KUKA KRL program: MyProgram_007().src

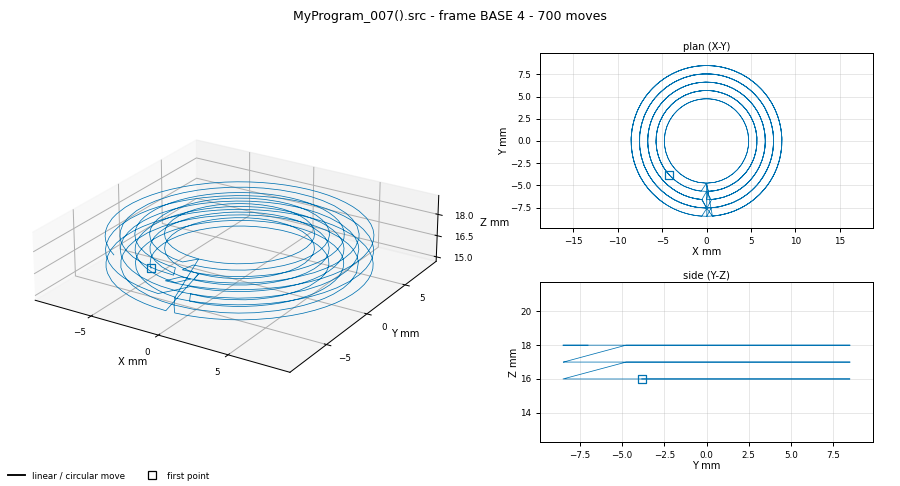
[picture p0: tool path of MyProgram_007().src in frame BASE 4, 700 of 700 moves have a stored position in this frame; points joined in program order, loops and branches not executed]
&ACCESS RVP
&REL 1
&PARAM TEMPLATE = C:\KRC\Roboter\Template\vorgabe
&PARAM EDITMASK = *
DEF MyProgram_007()
; ---- Setting reference (Base) ----
$BASE = BASE_DATA[4]

; --------------------------
; ---- Setting tool (TCP) ----
$TOOL = TOOL_DATA[3]
; --------------------------

$VEL.CP = VEL_APROX_PRINT
Startdeposition()
$VEL.CP = VEL_PRINT
LIN {X -4.1993,Y -3.8325,Z 16,A -3.0897,B 0,C 0,E1 0.1598,E2 90.0712} C_DIS
LIN {X -4.6903,Y -3.2125,Z 16,A -3.0815,B 0,C 0,E1 0.1598,E2 90.0712} C_DIS
LIN {X -5.0898,Y -2.5301,Z 16,A -3.0673,B 0,C 0,E1 0.1598,E2 90.0712} C_DIS
LIN {X -5.3905,Y -1.7989,Z 16,A -3.0475,B 0,C 0,E1 0.1598,E2 90.0712} C_DIS
LIN {X -5.5883,Y -1.0336,Z 16,A -3.0224,B 0,C 0,E1 0.1598,E2 90.0712} C_DIS
LIN {X -5.6777,Y -0.2482,Z 16,A -2.9925,B 0,C 0,E1 0.1598,E2 90.0712} C_DIS
LIN {X -5.6569,Y 0.542,Z 16,A -2.9584,B 0,C 0,E1 0.1598,E2 90.0713} C_DIS
LIN {X -5.5287,Y 1.3221,Z 16,A -2.9208,B 0,C 0,E1 0.1598,E2 90.0713} C_DIS
LIN {X -5.293,Y 2.077,Z 16,A -2.8803,B 0,C 0,E1 0.1598,E2 90.0714} C_DIS
LIN {X -4.954,Y 2.7915,Z 16,A -2.8378,B 0,C 0,E1 0.1598,E2 90.0715} C_DIS
LIN {X -4.5175,Y 3.4508,Z 16,A -2.7939,B 0,C 0,E1 0.1598,E2 90.0716} C_DIS
LIN {X -3.9945,Y 4.044,Z 16,A -2.7497,B 0,C 0,E1 0.1598,E2 90.0717} C_DIS
LIN {X -3.395,Y 4.5593,Z 16,A -2.7059,B 0,C 0,E1 0.1598,E2 90.0718} C_DIS
LIN {X -2.7289,Y 4.9855,Z 16,A -2.6634,B 0,C 0,E1 0.1598,E2 90.0719} C_DIS
LIN {X -2.0108,Y 5.316,Z 16,A -2.623,B 0,C 0,E1 0.1598,E2 90.072} C_DIS
LIN {X -1.2535,Y 5.5427,Z 16,A -2.5855,B 0,C 0,E1 0.1598,E2 90.0721} C_DIS
LIN {X -0.2754,Y 5.684,Z 16,A -2.5435,B 0,C 0,E1 0.1598,E2 90.0721} C_DIS
LIN {X 0.4673,Y 5.6661,Z 16,A -2.5168,B 0,C 0,E1 0.1598,E2 90.0722} C_DIS
LIN {X 1.1226,Y 5.5779,Z 16,A -2.4964,B 0,C 0,E1 0.1598,E2 90.0722} C_DIS
LIN {X 2.1788,Y 5.2504,Z 16,A -2.4712,B 0,C 0,E1 0.1598,E2 90.0722} C_DIS
LIN {X 2.8813,Y 4.8983,Z 16,A -2.4602,B 0,C 0,E1 0.1598,E2 90.0722} C_DIS
LIN {X 3.5298,Y 4.4549,Z 16,A -2.455,B 0,C 0,E1 0.1598,E2 90.0722} C_DIS
LIN {X 4.1099,Y 3.9251,Z 16,A -2.456,B 0,C 0,E1 0.1598,E2 90.0722} C_DIS
LIN {X 4.6118,Y 3.3208,Z 16,A -2.4631,B 0,C 0,E1 0.1598,E2 90.0721} C_DIS
LIN {X 5.0254,Y 2.653,Z 16,A -2.4761,B 0,C 0,E1 0.1598,E2 90.0721} C_DIS
LIN {X 5.3429,Y 1.9345,Z 16,A -2.4949,B 0,C 0,E1 0.1598,E2 90.0719} C_DIS
LIN {X 5.5612,Y 1.1798,Z 16,A -2.5188,B 0,C 0,E1 0.1598,E2 90.0719} C_DIS
LIN {X 5.6718,Y 0.4017,Z 16,A -2.5478,B 0,C 0,E1 0.1598,E2 90.0719} C_DIS
LIN {X 5.6312,Y -0.8177,Z 16,A -2.6006,B 0,C 0,E1 0.1598,E2 90.0713} C_DIS
LIN {X 5.4243,Y -1.7083,Z 16,A -2.6464,B 0,C 0,E1 0.1598,E2 90.0716} C_DIS
LIN {X 5.159,Y -2.3898,Z 16,A -2.6852,B 0,C 0,E1 0.1598,E2 90.0717} C_DIS
LIN {X 4.8093,Y -3.0322,Z 16,A -2.7254,B 0,C 0,E1 0.1598,E2 90.0717} C_DIS
LIN {X 4.3781,Y -3.6227,Z 16,A -2.7663,B 0,C 0,E1 0.1598,E2 90.0717} C_DIS
LIN {X 3.8775,Y -4.1555,Z 16,A -2.8073,B 0,C 0,E1 0.1598,E2 90.0717} C_DIS
LIN {X 3.3125,Y -4.6195,Z 16,A -2.8478,B 0,C 0,E1 0.1598,E2 90.0717} C_DIS
LIN {X 2.287,Y -5.2099,Z 16,A -2.9105,B 0,C 0,E1 0.1598,E2 90.0715} C_DIS
LIN {X 1.4913,Y -5.4882,Z 16,A -2.9516,B 0,C 0,E1 0.1598,E2 90.0716} C_DIS
LIN {X 0.8312,Y -5.6248,Z 16,A -2.9816,B 0,C 0,E1 0.1598,E2 90.0716} C_DIS
LIN {X -0.0092,Y -5.6859,Z 16,A -3.0151,B 0,C 0,E1 0.1598,E2 90.0716} C_DIS
Enddeposition()
LIN {X -0.0092,Y -5.6859,Z 16,A -3.0151,B 0,C 0,E1 0.1598,E2 90.0716} C_DIS
Startdeposition()
$VEL.CP = VEL_PRINT
LIN {X 0.5176,Y -6.5991,Z 16,A -3.034,B 0,C 0,E1 0.1598,E2 90.071} C_DIS
LIN {X 1.2141,Y -6.5071,Z 16,A -3.0051,B 0,C 0,E1 0.1598,E2 90.0715} C_DIS
LIN {X 1.897,Y -6.3414,Z 16,A -2.9731,B 0,C 0,E1 0.1598,E2 90.0715} C_DIS
LIN {X 2.5586,Y -6.1047,Z 16,A -2.9387,B 0,C 0,E1 0.1598,E2 90.0716} C_DIS
LIN {X 3.1928,Y -5.802,Z 16,A -2.9026,B 0,C 0,E1 0.1598,E2 90.0716} C_DIS
LIN {X 3.7886,Y -5.4294,Z 16,A -2.8649,B 0,C 0,E1 0.1598,E2 90.0716} C_DIS
LIN {X 4.3414,Y -4.9954,Z 16,A -2.8261,B 0,C 0,E1 0.1598,E2 90.0717} C_DIS
LIN {X 4.8479,Y -4.5083,Z 16,A -2.7868,B 0,C 0,E1 0.1598,E2 90.0717} C_DIS
LIN {X 5.2989,Y -3.9693,Z 16,A -2.7473,B 0,C 0,E1 0.1598,E2 90.0717} C_DIS
LIN {X 5.6898,Y -3.3855,Z 16,A -2.7081,B 0,C 0,E1 0.1598,E2 90.0717} C_DIS
LIN {X 6.0154,Y -2.7628,Z 16,A -2.6697,B 0,C 0,E1 0.1598,E2 90.0718} C_DIS
LIN {X 6.2743,Y -2.1096,Z 16,A -2.6324,B 0,C 0,E1 0.1598,E2 90.0718} C_DIS
LIN {X 6.4633,Y -1.4327,Z 16,A -2.5967,B 0,C 0,E1 0.1598,E2 90.0718} C_DIS
LIN {X 6.5765,Y -0.7393,Z 16,A -2.563,B 0,C 0,E1 0.1598,E2 90.0718} C_DIS
LIN {X 6.6202,Y -0.038,Z 16,A -2.5316,B 0,C 0,E1 0.1598,E2 90.0719} C_DIS
LIN {X 6.5859,Y 0.6639,Z 16,A -2.5031,B 0,C 0,E1 0.1598,E2 90.0719} C_DIS
LIN {X 6.4813,Y 1.3587,Z 16,A -2.4774,B 0,C 0,E1 0.1598,E2 90.0719} C_DIS
LIN {X 6.2989,Y 2.0375,Z 16,A -2.4553,B 0,C 0,E1 0.1598,E2 90.072} C_DIS
LIN {X 6.0478,Y 2.6938,Z 16,A -2.4367,B 0,C 0,E1 0.1598,E2 90.072} C_DIS
LIN {X 5.7274,Y 3.3193,Z 16,A -2.422,B 0,C 0,E1 0.1598,E2 90.0721} C_DIS
LIN {X 5.3436,Y 3.908,Z 16,A -2.4112,B 0,C 0,E1 0.1598,E2 90.0721} C_DIS
LIN {X 4.8987,Y 4.4518,Z 16,A -2.4046,B 0,C 0,E1 0.1598,E2 90.0721} C_DIS
LIN {X 4.3987,Y 4.9454,Z 16,A -2.4021,B 0,C 0,E1 0.1598,E2 90.0722} C_DIS
LIN {X 3.8499,Y 5.3843,Z 16,A -2.4038,B 0,C 0,E1 0.1598,E2 90.0722} C_DIS
LIN {X 2.9549,Y 5.9276,Z 16,A -2.4138,B 0,C 0,E1 0.1598,E2 90.0722} C_DIS
LIN {X 2.1433,Y 6.2629,Z 16,A -2.4296,B 0,C 0,E1 0.1598,E2 90.0722} C_DIS
LIN {X 1.4674,Y 6.4547,Z 16,A -2.4465,B 0,C 0,E1 0.1598,E2 90.0722} C_DIS
LIN {X 0.7748,Y 6.5728,Z 16,A -2.4671,B 0,C 0,E1 0.1598,E2 90.0722} C_DIS
LIN {X 0.0739,Y 6.6206,Z 16,A -2.4909,B 0,C 0,E1 0.1598,E2 90.0722} C_DIS
LIN {X -0.6281,Y 6.5907,Z 16,A -2.5181,B 0,C 0,E1 0.1598,E2 90.0722} C_DIS
LIN {X -1.3232,Y 6.4884,Z 16,A -2.5481,B 0,C 0,E1 0.1598,E2 90.0722} C_DIS
LIN {X -2.0031,Y 6.3109,Z 16,A -2.5806,B 0,C 0,E1 0.1598,E2 90.0722} C_DIS
LIN {X -2.6597,Y 6.0605,Z 16,A -2.6154,B 0,C 0,E1 0.1598,E2 90.0721} C_DIS
LIN {X -3.2875,Y 5.7451,Z 16,A -2.6518,B 0,C 0,E1 0.1598,E2 90.072} C_DIS
LIN {X -3.8778,Y 5.3647,Z 16,A -2.6896,B 0,C 0,E1 0.1598,E2 90.072} C_DIS
LIN {X -4.4251,Y 4.924,Z 16,A -2.7284,B 0,C 0,E1 0.1598,E2 90.0718} C_DIS
LIN {X -4.921,Y 4.4263,Z 16,A -2.7676,B 0,C 0,E1 0.1598,E2 90.0718} C_DIS
LIN {X -5.3638,Y 3.8808,Z 16,A -2.8069,B 0,C 0,E1 0.1598,E2 90.0717} C_DIS
LIN {X -5.745,Y 3.2907,Z 16,A -2.8458,B 0,C 0,E1 0.1598,E2 90.0717} C_DIS
LIN {X -6.0618,Y 2.6636,Z 16,A -2.8839,B 0,C 0,E1 0.1598,E2 90.0715} C_DIS
LIN {X -6.3071,Y 2.0053,Z 16,A -2.9206,B 0,C 0,E1 0.1598,E2 90.0715} C_DIS
LIN {X -6.4853,Y 1.3257,Z 16,A -2.9558,B 0,C 0,E1 0.1598,E2 90.0714} C_DIS
LIN {X -6.59,Y 0.631,Z 16,A -2.9889,B 0,C 0,E1 0.1598,E2 90.0714} C_DIS
LIN {X -6.6205,Y -0.0711,Z 16,A -3.0196,B 0,C 0,E1 0.1598,E2 90.0713} C_DIS
LIN {X -6.5747,Y -0.7722,Z 16,A -3.0475,B 0,C 0,E1 0.1598,E2 90.0713} C_DIS
LIN {X -6.4566,Y -1.4648,Z 16,A -3.0724,B 0,C 0,E1 0.1598,E2 90.0713} C_DIS
LIN {X -6.2639,Y -2.1405,Z 16,A -3.0938,B 0,C 0,E1 0.1598,E2 90.0713} C_DIS
LIN {X -6.001,Y -2.7921,Z 16,A -3.1116,B 0,C 0,E1 0.1598,E2 90.0713} C_DIS
LIN {X -5.5827,Y -3.5644,Z 16,A -3.1287,B 0,C 0,E1 0.1598,E2 90.071} C_DIS
LIN {X -4.9457,Y -4.3995,Z 16,A -3.1406,B 0,C 0,E1 0.1598,E2 90.071} C_DIS
LIN {X -4.4386,Y -4.9094,Z 16,A -3.1437,B 0,C 0,E1 0.1598,E2 90.0712} C_DIS
LIN {X -3.8804,Y -5.3625,Z 16,A -3.1424,B 0,C 0,E1 0.1598,E2 90.0712} C_DIS
LIN {X -3.2755,Y -5.7514,Z 16,A -3.1367,B 0,C 0,E1 0.1598,E2 90.0713} C_DIS
LIN {X -2.6323,Y -6.0729,Z 16,A -3.1267,B 0,C 0,E1 0.1598,E2 90.0713} C_DIS
LIN {X -1.9581,Y -6.3233,Z 16,A -3.1126,B 0,C 0,E1 0.1598,E2 90.0713} C_DIS
LIN {X -1.2608,Y -6.4991,Z 16,A -3.0945,B 0,C 0,E1 0.1598,E2 90.0714} C_DIS
LIN {X -0.5481,Y -6.5959,Z 16,A -3.0725,B 0,C 0,E1 0.1598,E2 90.0714} C_DIS
LIN {X -0.5481,Y -6.5959,Z 16,A -3.0725,B 0,C 0,E1 0.1598,E2 90.0714} C_DIS
Enddeposition()
LIN {X 0.0119,Y -7.5545,Z 16,A -3.0916,B 0,C 0,E1 0.1598,E2 90.0703} C_DIS
Startdeposition()
$VEL.CP = VEL_PRINT
LIN {X -0.9518,Y -7.4924,Z 16,A -3.1254,B 0,C 0,E1 0.1598,E2 90.0713} C_DIS
LIN {X -1.9009,Y -7.3137,Z 16,A -3.1527,B 0,C 0,E1 0.1598,E2 90.0713} C_DIS
LIN {X -2.9797,Y -6.9401,Z 16,A -3.1763,B 0,C 0,E1 0.1598,E2 90.0713} C_DIS
LIN {X -3.7254,Y -6.5689,Z 16,A -3.188,B 0,C 0,E1 0.1598,E2 90.0713} C_DIS
LIN {X -4.4267,Y -6.1193,Z 16,A -3.1947,B 0,C 0,E1 0.1598,E2 90.0713} C_DIS
LIN {X -5.0741,Y -5.5949,Z 16,A -3.1962,B 0,C 0,E1 0.1598,E2 90.0712} C_DIS
LIN {X -5.8749,Y -4.7558,Z 16,A -3.19,B 0,C 0,E1 0.1598,E2 90.071} C_DIS
LIN {X -6.5112,Y -3.8283,Z 16,A -3.174,B 0,C 0,E1 0.1598,E2 90.0708} C_DIS
LIN {X -6.9744,Y -2.9088,Z 16,A -3.1522,B 0,C 0,E1 0.1598,E2 90.0708} C_DIS
LIN {X -7.3358,Y -1.7986,Z 16,A -3.1185,B 0,C 0,E1 0.1598,E2 90.0708} C_DIS
LIN {X -7.5221,Y -0.731,Z 16,A -3.0803,B 0,C 0,E1 0.1598,E2 90.0708} C_DIS
LIN {X -7.5246,Y 0.7105,Z 16,A -3.0193,B 0,C 0,E1 0.1598,E2 90.0704} C_DIS
LIN {X -7.2713,Y 2.0637,Z 16,A -2.9531,B 0,C 0,E1 0.1598,E2 90.0707} C_DIS
LIN {X -6.8863,Y 3.1038,Z 16,A -2.8954,B 0,C 0,E1 0.1598,E2 90.0711} C_DIS
LIN {X -6.4131,Y 3.9965,Z 16,A -2.8405,B 0,C 0,E1 0.1598,E2 90.0713} C_DIS
LIN {X -5.7708,Y 4.8784,Z 16,A -2.7798,B 0,C 0,E1 0.1598,E2 90.0715} C_DIS
LIN {X -4.6762,Y 5.9363,Z 16,A -2.6947,B 0,C 0,E1 0.1598,E2 90.0715} C_DIS
LIN {X -3.8022,Y 6.5253,Z 16,A -2.638,B 0,C 0,E1 0.1598,E2 90.0719} C_DIS
LIN {X -2.7409,Y 7.0434,Z 16,A -2.577,B 0,C 0,E1 0.1598,E2 90.072} C_DIS
LIN {X -1.5757,Y 7.3865,Z 16,A -2.5196,B 0,C 0,E1 0.1598,E2 90.0722} C_DIS
LIN {X -0.8601,Y 7.5059,Z 16,A -2.4882,B 0,C 0,E1 0.1598,E2 90.0722} C_DIS
LIN {X 0.0453,Y 7.5578,Z 16,A -2.4526,B 0,C 0,E1 0.1598,E2 90.0722} C_DIS
LIN {X 1.3007,Y 7.4447,Z 16,A -2.411,B 0,C 0,E1 0.1598,E2 90.0723} C_DIS
LIN {X 2.297,Y 7.1992,Z 16,A -2.3846,B 0,C 0,E1 0.1598,E2 90.0723} C_DIS
LIN {X 3.4759,Y 6.7108,Z 16,A -2.3616,B 0,C 0,E1 0.1598,E2 90.0723} C_DIS
LIN {X 4.5236,Y 6.0538,Z 16,A -2.3507,B 0,C 0,E1 0.1598,E2 90.0722} C_DIS
LIN {X 5.2147,Y 5.4686,Z 16,A -2.3499,B 0,C 0,E1 0.1598,E2 90.0722} C_DIS
LIN {X 5.9309,Y 4.6831,Z 16,A -2.3567,B 0,C 0,E1 0.1598,E2 90.072} C_DIS
LIN {X 6.4566,Y 3.9262,Z 16,A -2.3695,B 0,C 0,E1 0.1598,E2 90.072} C_DIS
LIN {X 7.1647,Y 2.4074,Z 16,A -2.4069,B 0,C 0,E1 0.1598,E2 90.0711} C_DIS
LIN {X 7.4842,Y 1.0554,Z 16,A -2.4528,B 0,C 0,E1 0.1598,E2 90.0712} C_DIS
LIN {X 7.5583,Y 0.0222,Z 16,A -2.4944,B 0,C 0,E1 0.1598,E2 90.0716} C_DIS
LIN {X 7.4763,Y -1.08,Z 16,A -2.5442,B 0,C 0,E1 0.1598,E2 90.0715} C_DIS
LIN {X 7.317,Y -1.8715,Z 16,A -2.584,B 0,C 0,E1 0.1598,E2 90.0718} C_DIS
LIN {X 7.0768,Y -2.6424,Z 16,A -2.6256,B 0,C 0,E1 0.1598,E2 90.0718} C_DIS
LIN {X 6.7526,Y -3.3818,Z 16,A -2.669,B 0,C 0,E1 0.1598,E2 90.0718} C_DIS
LIN {X 6.3536,Y -4.0837,Z 16,A -2.7135,B 0,C 0,E1 0.1598,E2 90.0717} C_DIS
LIN {X 5.7553,Y -4.8965,Z 16,A -2.7699,B 0,C 0,E1 0.1598,E2 90.0715} C_DIS
LIN {X 4.7656,Y -5.867,Z 16,A -2.8474,B 0,C 0,E1 0.1598,E2 90.0713} C_DIS
LIN {X 3.9501,Y -6.4362,Z 16,A -2.9018,B 0,C 0,E1 0.1598,E2 90.0715} C_DIS
LIN {X 3.073,Y -6.9047,Z 16,A -2.9539,B 0,C 0,E1 0.1598,E2 90.0715} C_DIS
LIN {X 1.3721,Y -7.433,Z 16,A -3.0387,B 0,C 0,E1 0.1598,E2 90.0715} C_DIS
LIN {X 0.0119,Y -7.5545,Z 16,A -3.0938,B 0,C 0,E1 0.1598,E2 90.0715} C_DIS
Enddeposition()
LIN {X 0.0119,Y -7.5545,Z 16,A -3.0938,B 0,C 0,E1 0.1598,E2 90.0715} C_DIS
Startdeposition()
$VEL.CP = VEL_PRINT
LIN {X 0.6623,Y -8.4623,Z 16,A -3.1081,B 0,C 0,E1 0.1598,E2 90.0709} C_DIS
LIN {X 1.4918,Y -8.3555,Z 16,A -3.0737,B 0,C 0,E1 0.1598,E2 90.0714} C_DIS
LIN {X 2.3069,Y -8.1682,Z 16,A -3.0359,B 0,C 0,E1 0.1598,E2 90.0715} C_DIS
LIN {X 3.0995,Y -7.9014,Z 16,A -2.9955,B 0,C 0,E1 0.1598,E2 90.0715} C_DIS
LIN {X 3.8621,Y -7.558,Z 16,A -2.9529,B 0,C 0,E1 0.1598,E2 90.0715} C_DIS
LIN {X 4.5873,Y -7.1413,Z 16,A -2.9086,B 0,C 0,E1 0.1598,E2 90.0716} C_DIS
LIN {X 5.268,Y -6.6555,Z 16,A -2.863,B 0,C 0,E1 0.1598,E2 90.0716} C_DIS
LIN {X 6.0484,Y -5.96,Z 16,A -2.8046,B 0,C 0,E1 0.1598,E2 90.0716} C_DIS
LIN {X 6.8105,Y -5.064,Z 16,A -2.7384,B 0,C 0,E1 0.1598,E2 90.0715} C_DIS
LIN {X 7.2709,Y -4.3791,Z 16,A -2.6925,B 0,C 0,E1 0.1598,E2 90.0717} C_DIS
LIN {X 7.6619,Y -3.6523,Z 16,A -2.6472,B 0,C 0,E1 0.1598,E2 90.0717} C_DIS
LIN {X 7.9811,Y -2.8913,Z 16,A -2.6031,B 0,C 0,E1 0.1598,E2 90.0717} C_DIS
LIN {X 8.224,Y -2.1025,Z 16,A -2.5606,B 0,C 0,E1 0.1598,E2 90.0718} C_DIS
LIN {X 8.3896,Y -1.2939,Z 16,A -2.5201,B 0,C 0,E1 0.1598,E2 90.0718} C_DIS
LIN {X 8.4751,Y -0.473,Z 16,A -2.482,B 0,C 0,E1 0.1598,E2 90.0718} C_DIS
LIN {X 8.4802,Y 0.3524,Z 16,A -2.4467,B 0,C 0,E1 0.1598,E2 90.0719} C_DIS
LIN {X 8.4047,Y 1.1742,Z 16,A -2.4145,B 0,C 0,E1 0.1598,E2 90.0719} C_DIS
LIN {X 8.2506,Y 1.9849,Z 16,A -2.3858,B 0,C 0,E1 0.1598,E2 90.072} C_DIS
LIN {X 8.019,Y 2.777,Z 16,A -2.3606,B 0,C 0,E1 0.1598,E2 90.072} C_DIS
LIN {X 7.7115,Y 3.5429,Z 16,A -2.3395,B 0,C 0,E1 0.1598,E2 90.0721} C_DIS
LIN {X 7.3312,Y 4.2754,Z 16,A -2.3224,B 0,C 0,E1 0.1598,E2 90.0721} C_DIS
LIN {X 6.8816,Y 4.9676,Z 16,A -2.3096,B 0,C 0,E1 0.1598,E2 90.0722} C_DIS
LIN {X 6.367,Y 5.613,Z 16,A -2.3013,B 0,C 0,E1 0.1598,E2 90.0722} C_DIS
LIN {X 5.6415,Y 6.3466,Z 16,A -2.2968,B 0,C 0,E1 0.1598,E2 90.0722} C_DIS
LIN {X 4.7819,Y 7.0135,Z 16,A -2.3004,B 0,C 0,E1 0.1598,E2 90.0722} C_DIS
LIN {X 4.0293,Y 7.4733,Z 16,A -2.3088,B 0,C 0,E1 0.1598,E2 90.0723} C_DIS
LIN {X 2.9445,Y 7.9626,Z 16,A -2.3281,B 0,C 0,E1 0.1598,E2 90.0723} C_DIS
LIN {X 2.1419,Y 8.2149,Z 16,A -2.3472,B 0,C 0,E1 0.1598,E2 90.0723} C_DIS
LIN {X 1.3183,Y 8.3862,Z 16,A -2.3704,B 0,C 0,E1 0.1598,E2 90.0723} C_DIS
LIN {X 0.4817,Y 8.4746,Z 16,A -2.3976,B 0,C 0,E1 0.1598,E2 90.0723} C_DIS
LIN {X -0.3594,Y 8.4792,Z 16,A -2.4285,B 0,C 0,E1 0.1598,E2 90.0723} C_DIS
LIN {X -1.1968,Y 8.4012,Z 16,A -2.4627,B 0,C 0,E1 0.1598,E2 90.0723} C_DIS
LIN {X -2.0225,Y 8.2411,Z 16,A -2.4999,B 0,C 0,E1 0.1598,E2 90.0723} C_DIS
LIN {X -2.8283,Y 8.0002,Z 16,A -2.5398,B 0,C 0,E1 0.1598,E2 90.0722} C_DIS
LIN {X -3.6063,Y 7.6809,Z 16,A -2.582,B 0,C 0,E1 0.1598,E2 90.0721} C_DIS
LIN {X -4.3488,Y 7.2859,Z 16,A -2.626,B 0,C 0,E1 0.1598,E2 90.072} C_DIS
LIN {X -5.049,Y 6.8199,Z 16,A -2.6715,B 0,C 0,E1 0.1598,E2 90.072} C_DIS
LIN {X -5.6995,Y 6.2869,Z 16,A -2.7179,B 0,C 0,E1 0.1598,E2 90.0718} C_DIS
LIN {X -6.2942,Y 5.6921,Z 16,A -2.7648,B 0,C 0,E1 0.1598,E2 90.0718} C_DIS
LIN {X -6.827,Y 5.0413,Z 16,A -2.8118,B 0,C 0,E1 0.1598,E2 90.0716} C_DIS
LIN {X -7.2932,Y 4.3411,Z 16,A -2.8585,B 0,C 0,E1 0.1598,E2 90.0716} C_DIS
LIN {X -7.7769,Y 3.4075,Z 16,A -2.9153,B 0,C 0,E1 0.1598,E2 90.0712} C_DIS
LIN {X -8.1287,Y 2.4526,Z 16,A -2.9685,B 0,C 0,E1 0.1598,E2 90.0712} C_DIS
LIN {X -8.3775,Y 1.3673,Z 16,A -3.0232,B 0,C 0,E1 0.1598,E2 90.0709} C_DIS
LIN {X -8.4835,Y 0.3842,Z 16,A -3.0685,B 0,C 0,E1 0.1598,E2 90.0709} C_DIS
LIN {X -8.4591,Y -0.7483,Z 16,A -3.1153,B 0,C 0,E1 0.1598,E2 90.0708} C_DIS
LIN {X -8.3086,Y -1.7475,Z 16,A -3.1519,B 0,C 0,E1 0.1598,E2 90.0708} C_DIS
LIN {X -8.007,Y -2.8254,Z 16,A -3.1862,B 0,C 0,E1 0.1598,E2 90.0708} C_DIS
LIN {X -7.5834,Y -3.8091,Z 16,A -3.2122,B 0,C 0,E1 0.1598,E2 90.0708} C_DIS
LIN {X -7.1612,Y -4.5547,Z 16,A -3.2284,B 0,C 0,E1 0.1598,E2 90.071} C_DIS
LIN {X -6.6657,Y -5.2537,Z 16,A -3.2397,B 0,C 0,E1 0.1598,E2 90.071} C_DIS
LIN {X -6.1026,Y -5.8995,Z 16,A -3.2463,B 0,C 0,E1 0.1598,E2 90.071} C_DIS
LIN {X -5.2057,Y -6.7068,Z 16,A -3.2474,B 0,C 0,E1 0.1598,E2 90.071} C_DIS
LIN {X -4.4325,Y -7.2404,Z 16,A -3.2418,B 0,C 0,E1 0.1598,E2 90.0711} C_DIS
LIN {X -3.7745,Y -7.6036,Z 16,A -3.2331,B 0,C 0,E1 0.1598,E2 90.0711} C_DIS
LIN {X -3.0867,Y -7.9065,Z 16,A -3.2207,B 0,C 0,E1 0.1598,E2 90.0712} C_DIS
LIN {X -2.3753,Y -8.1484,Z 16,A -3.2049,B 0,C 0,E1 0.1598,E2 90.0712} C_DIS
LIN {X -1.6454,Y -8.3273,Z 16,A -3.1858,B 0,C 0,E1 0.1598,E2 90.0713} C_DIS
LIN {X -0.9025,Y -8.4402,Z 16,A -3.1633,B 0,C 0,E1 0.1598,E2 90.0713} C_DIS
LIN {X 0.0356,Y -8.4913,Z 16,A -3.1311,B 0,C 0,E1 0.1598,E2 90.0713} C_DIS
Enddeposition()
LIN {X 0.0003,Y -4.7569,Z 17,A -2.9589,B 0,C 0,E1 0.1598,E2 90.0603} C_DIS
Startdeposition()
$VEL.CP = VEL_PRINT
LIN {X 0.0003,Y -4.7569,Z 17,A -2.9646,B 0,C 0,E1 0.1598,E2 90.0661} C_DIS
LIN {X -0.9154,Y -4.6636,Z 17,A -2.9991,B 0,C 0,E1 0.1598,E2 90.0709} C_DIS
LIN {X -1.6245,Y -4.4647,Z 17,A -3.0173,B 0,C 0,E1 0.1598,E2 90.0715} C_DIS
LIN {X -2.2939,Y -4.158,Z 17,A -3.0289,B 0,C 0,E1 0.1598,E2 90.0715} C_DIS
LIN {X -2.9104,Y -3.7559,Z 17,A -3.0345,B 0,C 0,E1 0.1598,E2 90.0715} C_DIS
LIN {X -3.4563,Y -3.2615,Z 17,A -3.0336,B 0,C 0,E1 0.1598,E2 90.0714} C_DIS
LIN {X -3.9175,Y -2.6875,Z 17,A -3.0263,B 0,C 0,E1 0.1598,E2 90.0714} C_DIS
LIN {X -4.2861,Y -2.05,Z 17,A -3.0129,B 0,C 0,E1 0.1598,E2 90.0714} C_DIS
LIN {X -4.5515,Y -1.3631,Z 17,A -2.9936,B 0,C 0,E1 0.1598,E2 90.0714} C_DIS
LIN {X -4.7058,Y -0.6432,Z 17,A -2.9688,B 0,C 0,E1 0.1598,E2 90.0714} C_DIS
LIN {X -4.7514,Y 0.0918,Z 17,A -2.9395,B 0,C 0,E1 0.1598,E2 90.0714} C_DIS
LIN {X -4.6778,Y 0.8245,Z 17,A -2.9058,B 0,C 0,E1 0.1598,E2 90.0714} C_DIS
LIN {X -4.496,Y 1.538,Z 17,A -2.869,B 0,C 0,E1 0.1598,E2 90.0714} C_DIS
LIN {X -4.2028,Y 2.2133,Z 17,A -2.8298,B 0,C 0,E1 0.1598,E2 90.0716} C_DIS
LIN {X -3.8104,Y 2.836,Z 17,A -2.7891,B 0,C 0,E1 0.1598,E2 90.0716} C_DIS
LIN {X -3.326,Y 3.3904,Z 17,A -2.7479,B 0,C 0,E1 0.1598,E2 90.0718} C_DIS
LIN {X -2.762,Y 3.8634,Z 17,A -2.7072,B 0,C 0,E1 0.1598,E2 90.0718} C_DIS
LIN {X -2.1333,Y 4.2469,Z 17,A -2.6678,B 0,C 0,E1 0.1598,E2 90.0719} C_DIS
LIN {X -1.4507,Y 4.5231,Z 17,A -2.631,B 0,C 0,E1 0.1598,E2 90.072} C_DIS
LIN {X -0.734,Y 4.6918,Z 17,A -2.5975,B 0,C 0,E1 0.1598,E2 90.072} C_DIS
LIN {X -0.0003,Y 4.75,Z 17,A -2.568,B 0,C 0,E1 0.1598,E2 90.0721} C_DIS
LIN {X 0.7335,Y 4.6929,Z 17,A -2.5434,B 0,C 0,E1 0.1598,E2 90.0721} C_DIS
LIN {X 1.4499,Y 4.5234,Z 17,A -2.5241,B 0,C 0,E1 0.1598,E2 90.0721} C_DIS
LIN {X 2.1318,Y 4.246,Z 17,A -2.5107,B 0,C 0,E1 0.1598,E2 90.0721} C_DIS
LIN {X 2.7629,Y 3.8665,Z 17,A -2.5034,B 0,C 0,E1 0.1598,E2 90.0721} C_DIS
LIN {X 3.3252,Y 3.3912,Z 17,A -2.5028,B 0,C 0,E1 0.1598,E2 90.0721} C_DIS
LIN {X 3.809,Y 2.8365,Z 17,A -2.5084,B 0,C 0,E1 0.1598,E2 90.0721} C_DIS
LIN {X 4.2027,Y 2.2144,Z 17,A -2.5203,B 0,C 0,E1 0.1598,E2 90.072} C_DIS
LIN {X 4.4932,Y 1.538,Z 17,A -2.5382,B 0,C 0,E1 0.1598,E2 90.072} C_DIS
LIN {X 4.6765,Y 0.825,Z 17,A -2.5617,B 0,C 0,E1 0.1598,E2 90.0719} C_DIS
LIN {X 4.7489,Y 0.0927,Z 17,A -2.5901,B 0,C 0,E1 0.1598,E2 90.0719} C_DIS
LIN {X 4.7075,Y -0.6423,Z 17,A -2.6228,B 0,C 0,E1 0.1598,E2 90.0718} C_DIS
LIN {X 4.5519,Y -1.3622,Z 17,A -2.6591,B 0,C 0,E1 0.1598,E2 90.0718} C_DIS
LIN {X 4.2854,Y -2.0486,Z 17,A -2.698,B 0,C 0,E1 0.1598,E2 90.0718} C_DIS
LIN {X 3.9169,Y -2.6859,Z 17,A -2.7387,B 0,C 0,E1 0.1598,E2 90.0718} C_DIS
LIN {X 3.4549,Y -3.2589,Z 17,A -2.78,B 0,C 0,E1 0.1598,E2 90.0718} C_DIS
LIN {X 2.91,Y -3.7538,Z 17,A -2.8211,B 0,C 0,E1 0.1598,E2 90.0717} C_DIS
LIN {X 2.2944,Y -4.1575,Z 17,A -2.8608,B 0,C 0,E1 0.1598,E2 90.0717} C_DIS
LIN {X 1.6248,Y -4.4628,Z 17,A -2.8984,B 0,C 0,E1 0.1598,E2 90.0717} C_DIS
LIN {X 0.9157,Y -4.6613,Z 17,A -2.9329,B 0,C 0,E1 0.1598,E2 90.0717} C_DIS
LIN {X 0.0003,Y -4.7569,Z 17,A -2.9705,B 0,C 0,E1 0.1598,E2 90.0717} C_DIS
Enddeposition()
LIN {X 0.0003,Y -4.7569,Z 17,A -2.9705,B 0,C 0,E1 0.1598,E2 90.0717} C_DIS
Startdeposition()
$VEL.CP = VEL_PRINT
LIN {X 0.2128,Y -5.6787,Z 17,A -3.0014,B 0,C 0,E1 0.1598,E2 90.071} C_DIS
LIN {X 1.0465,Y -5.5847,Z 17,A -2.9673,B 0,C 0,E1 0.1598,E2 90.0716} C_DIS
LIN {X 1.8578,Y -5.3707,Z 17,A -2.9285,B 0,C 0,E1 0.1598,E2 90.0716} C_DIS
LIN {X 2.6285,Y -5.0388,Z 17,A -2.8861,B 0,C 0,E1 0.1598,E2 90.0716} C_DIS
LIN {X 3.3423,Y -4.5975,Z 17,A -2.8411,B 0,C 0,E1 0.1598,E2 90.0716} C_DIS
LIN {X 3.9821,Y -4.0543,Z 17,A -2.7945,B 0,C 0,E1 0.1598,E2 90.0717} C_DIS
LIN {X 4.5363,Y -3.4241,Z 17,A -2.7473,B 0,C 0,E1 0.1598,E2 90.0717} C_DIS
LIN {X 4.9923,Y -2.7193,Z 17,A -2.7006,B 0,C 0,E1 0.1598,E2 90.0717} C_DIS
LIN {X 5.3382,Y -1.9545,Z 17,A -2.6553,B 0,C 0,E1 0.1598,E2 90.0717} C_DIS
LIN {X 5.5684,Y -1.1471,Z 17,A -2.6125,B 0,C 0,E1 0.1598,E2 90.0717} C_DIS
LIN {X 5.6762,Y -0.3146,Z 17,A -2.5732,B 0,C 0,E1 0.1598,E2 90.0717} C_DIS
LIN {X 5.6593,Y 0.5246,Z 17,A -2.5382,B 0,C 0,E1 0.1598,E2 90.0717} C_DIS
LIN {X 5.5198,Y 1.352,Z 17,A -2.5082,B 0,C 0,E1 0.1598,E2 90.0718} C_DIS
LIN {X 5.2598,Y 2.1498,Z 17,A -2.4839,B 0,C 0,E1 0.1598,E2 90.0718} C_DIS
LIN {X 4.8853,Y 2.9006,Z 17,A -2.4659,B 0,C 0,E1 0.1598,E2 90.072} C_DIS
LIN {X 4.4057,Y 3.589,Z 17,A -2.4544,B 0,C 0,E1 0.1598,E2 90.072} C_DIS
LIN {X 3.8296,Y 4.1992,Z 17,A -2.4499,B 0,C 0,E1 0.1598,E2 90.072} C_DIS
LIN {X 3.1694,Y 4.7172,Z 17,A -2.4523,B 0,C 0,E1 0.1598,E2 90.0721} C_DIS
LIN {X 2.4404,Y 5.1328,Z 17,A -2.4617,B 0,C 0,E1 0.1598,E2 90.0721} C_DIS
LIN {X 1.6577,Y 5.4359,Z 17,A -2.4777,B 0,C 0,E1 0.1598,E2 90.0722} C_DIS
LIN {X 0.8391,Y 5.6203,Z 17,A -2.5002,B 0,C 0,E1 0.1598,E2 90.0722} C_DIS
LIN {X 0.0024,Y 5.682,Z 17,A -2.5284,B 0,C 0,E1 0.1598,E2 90.0722} C_DIS
LIN {X -0.8342,Y 5.6197,Z 17,A -2.5619,B 0,C 0,E1 0.1598,E2 90.0722} C_DIS
LIN {X -1.6532,Y 5.4372,Z 17,A -2.5998,B 0,C 0,E1 0.1598,E2 90.0721} C_DIS
LIN {X -2.4353,Y 5.1333,Z 17,A -2.6415,B 0,C 0,E1 0.1598,E2 90.0721} C_DIS
LIN {X -3.1667,Y 4.7217,Z 17,A -2.6858,B 0,C 0,E1 0.1598,E2 90.0719} C_DIS
LIN {X -3.7548,Y 4.2748,Z 17,A -2.7263,B 0,C 0,E1 0.1598,E2 90.0718} C_DIS
LIN {X -4.4171,Y 3.5762,Z 17,A -2.7801,B 0,C 0,E1 0.1598,E2 90.0716} C_DIS
LIN {X -4.8614,Y 2.947,Z 17,A -2.823,B 0,C 0,E1 0.1598,E2 90.0716} C_DIS
LIN {X -5.2149,Y 2.2626,Z 17,A -2.8648,B 0,C 0,E1 0.1598,E2 90.0716} C_DIS
LIN {X -5.4728,Y 1.5369,Z 17,A -2.9049,B 0,C 0,E1 0.1598,E2 90.0714} C_DIS
LIN {X -5.6309,Y 0.7831,Z 17,A -2.9425,B 0,C 0,E1 0.1598,E2 90.0714} C_DIS
LIN {X -5.6854,Y 0.0147,Z 17,A -2.9769,B 0,C 0,E1 0.1598,E2 90.0714} C_DIS
LIN {X -5.6349,Y -0.7538,Z 17,A -3.0074,B 0,C 0,E1 0.1598,E2 90.0713} C_DIS
LIN {X -5.4819,Y -1.5088,Z 17,A -3.0337,B 0,C 0,E1 0.1598,E2 90.0713} C_DIS
LIN {X -5.2259,Y -2.2353,Z 17,A -3.055,B 0,C 0,E1 0.1598,E2 90.0713} C_DIS
LIN {X -4.8752,Y -2.9208,Z 17,A -3.071,B 0,C 0,E1 0.1598,E2 90.0713} C_DIS
LIN {X -4.4354,Y -3.5528,Z 17,A -3.0816,B 0,C 0,E1 0.1598,E2 90.0713} C_DIS
LIN {X -3.9149,Y -4.1203,Z 17,A -3.0865,B 0,C 0,E1 0.1598,E2 90.0713} C_DIS
LIN {X -3.3226,Y -4.6126,Z 17,A -3.0856,B 0,C 0,E1 0.1598,E2 90.0713} C_DIS
LIN {X -2.4989,Y -5.1111,Z 17,A -3.0765,B 0,C 0,E1 0.1598,E2 90.0713} C_DIS
LIN {X -1.4941,Y -5.4855,Z 17,A -3.0555,B 0,C 0,E1 0.1598,E2 90.0714} C_DIS
LIN {X -0.8359,Y -5.6251,Z 17,A -3.0373,B 0,C 0,E1 0.1598,E2 90.0715} C_DIS
LIN {X 0.0029,Y -5.6863,Z 17,A -3.0092,B 0,C 0,E1 0.1598,E2 90.0715} C_DIS
Enddeposition()
LIN {X 0.0029,Y -5.6863,Z 17,A -3.0092,B 0,C 0,E1 0.1598,E2 90.0715} C_DIS
Startdeposition()
$VEL.CP = VEL_PRINT
LIN {X -0.5105,Y -6.5987,Z 17,A -3.0663,B 0,C 0,E1 0.1598,E2 90.0709} C_DIS
LIN {X -1.2181,Y -6.506,Z 17,A -3.0888,B 0,C 0,E1 0.1598,E2 90.0714} C_DIS
LIN {X -1.9118,Y -6.3376,Z 17,A -3.1071,B 0,C 0,E1 0.1598,E2 90.0714} C_DIS
LIN {X -2.5826,Y -6.094,Z 17,A -3.1214,B 0,C 0,E1 0.1598,E2 90.0714} C_DIS
LIN {X -3.2243,Y -5.7814,Z 17,A -3.1317,B 0,C 0,E1 0.1598,E2 90.0714} C_DIS
LIN {X -3.8273,Y -5.3994,Z 17,A -3.1377,B 0,C 0,E1 0.1598,E2 90.0714} C_DIS
LIN {X -4.3866,Y -4.956,Z 17,A -3.1394,B 0,C 0,E1 0.1598,E2 90.0713} C_DIS
LIN {X -4.8946,Y -4.4547,Z 17,A -3.1368,B 0,C 0,E1 0.1598,E2 90.0713} C_DIS
LIN {X -5.3462,Y -3.9021,Z 17,A -3.1301,B 0,C 0,E1 0.1598,E2 90.0713} C_DIS
LIN {X -5.7362,Y -3.3042,Z 17,A -3.1191,B 0,C 0,E1 0.1598,E2 90.0713} C_DIS
LIN {X -6.0592,Y -2.6676,Z 17,A -3.1041,B 0,C 0,E1 0.1598,E2 90.0713} C_DIS
LIN {X -6.3103,Y -1.9994,Z 17,A -3.0851,B 0,C 0,E1 0.1598,E2 90.0713} C_DIS
LIN {X -6.4886,Y -1.3082,Z 17,A -3.0625,B 0,C 0,E1 0.1598,E2 90.0713} C_DIS
LIN {X -6.5908,Y -0.6019,Z 17,A -3.0364,B 0,C 0,E1 0.1598,E2 90.0713} C_DIS
LIN {X -6.6203,Y 0.1113,Z 17,A -3.0074,B 0,C 0,E1 0.1598,E2 90.0713} C_DIS
LIN {X -6.5691,Y 0.8232,Z 17,A -2.9755,B 0,C 0,E1 0.1598,E2 90.0713} C_DIS
LIN {X -6.4418,Y 1.5256,Z 17,A -2.9412,B 0,C 0,E1 0.1598,E2 90.0713} C_DIS
LIN {X -6.2407,Y 2.2106,Z 17,A -2.905,B 0,C 0,E1 0.1598,E2 90.0715} C_DIS
LIN {X -5.9677,Y 2.8701,Z 17,A -2.8671,B 0,C 0,E1 0.1598,E2 90.0715} C_DIS
LIN {X -5.6208,Y 3.494,Z 17,A -2.8281,B 0,C 0,E1 0.1598,E2 90.0716} C_DIS
LIN {X -5.2117,Y 4.0788,Z 17,A -2.7884,B 0,C 0,E1 0.1598,E2 90.0716} C_DIS
LIN {X -4.7429,Y 4.617,Z 17,A -2.7484,B 0,C 0,E1 0.1598,E2 90.0718} C_DIS
LIN {X -4.2187,Y 5.1012,Z 17,A -2.7087,B 0,C 0,E1 0.1598,E2 90.0718} C_DIS
LIN {X -3.6446,Y 5.5252,Z 17,A -2.6697,B 0,C 0,E1 0.1598,E2 90.0719} C_DIS
LIN {X -3.0288,Y 5.886,Z 17,A -2.6318,B 0,C 0,E1 0.1598,E2 90.072} C_DIS
LIN {X -2.378,Y 6.1791,Z 17,A -2.5954,B 0,C 0,E1 0.1598,E2 90.072} C_DIS
LIN {X -1.6993,Y 6.4002,Z 17,A -2.561,B 0,C 0,E1 0.1598,E2 90.0721} C_DIS
LIN {X -1.0004,Y 6.5451,Z 17,A -2.5291,B 0,C 0,E1 0.1598,E2 90.0721} C_DIS
LIN {X -0.1114,Y 6.6225,Z 17,A -2.4931,B 0,C 0,E1 0.1598,E2 90.0722} C_DIS
LIN {X 0.9415,Y 6.5527,Z 17,A -2.4572,B 0,C 0,E1 0.1598,E2 90.0722} C_DIS
LIN {X 1.6677,Y 6.4067,Z 17,A -2.4365,B 0,C 0,E1 0.1598,E2 90.0723} C_DIS
LIN {X 2.3728,Y 6.1794,Z 17,A -2.4201,B 0,C 0,E1 0.1598,E2 90.0723} C_DIS
LIN {X 3.0479,Y 5.8746,Z 17,A -2.4081,B 0,C 0,E1 0.1598,E2 90.0723} C_DIS
LIN {X 3.6849,Y 5.4968,Z 17,A -2.4006,B 0,C 0,E1 0.1598,E2 90.0723} C_DIS
LIN {X 4.2766,Y 5.0512,Z 17,A -2.3976,B 0,C 0,E1 0.1598,E2 90.0723} C_DIS
LIN {X 4.8153,Y 4.5426,Z 17,A -2.3992,B 0,C 0,E1 0.1598,E2 90.0723} C_DIS
LIN {X 5.2934,Y 3.9769,Z 17,A -2.4056,B 0,C 0,E1 0.1598,E2 90.0722} C_DIS
LIN {X 5.7029,Y 3.3595,Z 17,A -2.4166,B 0,C 0,E1 0.1598,E2 90.0722} C_DIS
LIN {X 6.0433,Y 2.7015,Z 17,A -2.432,B 0,C 0,E1 0.1598,E2 90.0721} C_DIS
LIN {X 6.3076,Y 2.0094,Z 17,A -2.4516,B 0,C 0,E1 0.1598,E2 90.0721} C_DIS
LIN {X 6.4909,Y 1.2917,Z 17,A -2.4753,B 0,C 0,E1 0.1598,E2 90.072} C_DIS
LIN {X 6.5941,Y 0.5583,Z 17,A -2.5026,B 0,C 0,E1 0.1598,E2 90.072} C_DIS
LIN {X 6.616,Y -0.182,Z 17,A -2.5333,B 0,C 0,E1 0.1598,E2 90.0719} C_DIS
LIN {X 6.5559,Y -0.9204,Z 17,A -2.5668,B 0,C 0,E1 0.1598,E2 90.0719} C_DIS
LIN {X 6.4112,Y -1.647,Z 17,A -2.603,B 0,C 0,E1 0.1598,E2 90.0719} C_DIS
LIN {X 6.1871,Y -2.353,Z 17,A -2.6413,B 0,C 0,E1 0.1598,E2 90.0718} C_DIS
LIN {X 5.8863,Y -3.0299,Z 17,A -2.6811,B 0,C 0,E1 0.1598,E2 90.0718} C_DIS
LIN {X 5.511,Y -3.6685,Z 17,A -2.7221,B 0,C 0,E1 0.1598,E2 90.0718} C_DIS
LIN {X 5.0653,Y -4.2602,Z 17,A -2.7636,B 0,C 0,E1 0.1598,E2 90.0718} C_DIS
LIN {X 4.5567,Y -4.7987,Z 17,A -2.8052,B 0,C 0,E1 0.1598,E2 90.0717} C_DIS
LIN {X 3.9921,Y -5.2781,Z 17,A -2.8463,B 0,C 0,E1 0.1598,E2 90.0717} C_DIS
LIN {X 3.3775,Y -5.6913,Z 17,A -2.8865,B 0,C 0,E1 0.1598,E2 90.0717} C_DIS
LIN {X 2.7211,Y -6.0348,Z 17,A -2.9251,B 0,C 0,E1 0.1598,E2 90.0717} C_DIS
LIN {X 2.0296,Y -6.3006,Z 17,A -2.9618,B 0,C 0,E1 0.1598,E2 90.0716} C_DIS
LIN {X 1.3127,Y -6.487,Z 17,A -2.996,B 0,C 0,E1 0.1598,E2 90.0716} C_DIS
LIN {X 0.5797,Y -6.5949,Z 17,A -3.0275,B 0,C 0,E1 0.1598,E2 90.0716} C_DIS
LIN {X 0.5797,Y -6.5949,Z 17,A -3.0275,B 0,C 0,E1 0.1598,E2 90.0716} C_DIS
Enddeposition()
LIN {X 0.0486,Y -7.5544,Z 17,A -3.0867,B 0,C 0,E1 0.1598,E2 90.0703} C_DIS
Startdeposition()
$VEL.CP = VEL_PRINT
LIN {X 0.9086,Y -7.5022,Z 17,A -3.054,B 0,C 0,E1 0.1598,E2 90.0714} C_DIS
LIN {X 2.0271,Y -7.2761,Z 17,A -3.0035,B 0,C 0,E1 0.1598,E2 90.0715} C_DIS
LIN {X 2.8194,Y -7.0071,Z 17,A -2.963,B 0,C 0,E1 0.1598,E2 90.0715} C_DIS
LIN {X 3.894,Y -6.4765,Z 17,A -2.9009,B 0,C 0,E1 0.1598,E2 90.0715} C_DIS
LIN {X 4.7584,Y -5.8657,Z 17,A -2.8432,B 0,C 0,E1 0.1598,E2 90.0716} C_DIS
LIN {X 5.3842,Y -5.2954,Z 17,A -2.796,B 0,C 0,E1 0.1598,E2 90.0716} C_DIS
LIN {X 5.9429,Y -4.6593,Z 17,A -2.7484,B 0,C 0,E1 0.1598,E2 90.0717} C_DIS
LIN {X 6.7846,Y -3.3273,Z 17,A -2.66,B 0,C 0,E1 0.1598,E2 90.0709} C_DIS
LIN {X 7.243,Y -2.1442,Z 17,A -2.5932,B 0,C 0,E1 0.1598,E2 90.0713} C_DIS
LIN {X 7.4326,Y -1.3418,Z 17,A -2.5525,B 0,C 0,E1 0.1598,E2 90.0718} C_DIS
LIN {X 7.5327,Y -0.5236,Z 17,A -2.514,B 0,C 0,E1 0.1598,E2 90.0718} C_DIS
LIN {X 7.5399,Y 0.5068,Z 17,A -2.4696,B 0,C 0,E1 0.1598,E2 90.0716} C_DIS
LIN {X 7.4027,Y 1.5184,Z 17,A -2.4318,B 0,C 0,E1 0.1598,E2 90.0717} C_DIS
LIN {X 7.1531,Y 2.4423,Z 17,A -2.4018,B 0,C 0,E1 0.1598,E2 90.0718} C_DIS
LIN {X 6.603,Y 3.6743,Z 17,A -2.3695,B 0,C 0,E1 0.1598,E2 90.0716} C_DIS
LIN {X 6.1561,Y 4.3834,Z 17,A -2.3564,B 0,C 0,E1 0.1598,E2 90.0721} C_DIS
LIN {X 5.4053,Y 5.2814,Z 17,A -2.3458,B 0,C 0,E1 0.1598,E2 90.072} C_DIS
LIN {X 4.6862,Y 5.9239,Z 17,A -2.3453,B 0,C 0,E1 0.1598,E2 90.0722} C_DIS
LIN {X 3.5934,Y 6.6476,Z 17,A -2.3549,B 0,C 0,E1 0.1598,E2 90.0721} C_DIS
LIN {X 2.4904,Y 7.1355,Z 17,A -2.3751,B 0,C 0,E1 0.1598,E2 90.0722} C_DIS
LIN {X 1.4199,Y 7.4185,Z 17,A -2.4028,B 0,C 0,E1 0.1598,E2 90.0723} C_DIS
LIN {X 0.5416,Y 7.5351,Z 17,A -2.4303,B 0,C 0,E1 0.1598,E2 90.0723} C_DIS
LIN {X -0.3443,Y 7.5454,Z 17,A -2.4626,B 0,C 0,E1 0.1598,E2 90.0723} C_DIS
LIN {X -1.4443,Y 7.4182,Z 17,A -2.5085,B 0,C 0,E1 0.1598,E2 90.0723} C_DIS
LIN {X -2.3141,Y 7.1938,Z 17,A -2.5501,B 0,C 0,E1 0.1598,E2 90.0722} C_DIS
LIN {X -3.4213,Y 6.7335,Z 17,A -2.6103,B 0,C 0,E1 0.1598,E2 90.072} C_DIS
LIN {X -4.1863,Y 6.2865,Z 17,A -2.6574,B 0,C 0,E1 0.1598,E2 90.072} C_DIS
LIN {X -5.144,Y 5.5358,Z 17,A -2.7242,B 0,C 0,E1 0.1598,E2 90.0717} C_DIS
LIN {X -5.8664,Y 4.7573,Z 17,A -2.7836,B 0,C 0,E1 0.1598,E2 90.0716} C_DIS
LIN {X -6.3634,Y 4.0682,Z 17,A -2.831,B 0,C 0,E1 0.1598,E2 90.0716} C_DIS
LIN {X -6.9694,Y 2.9206,Z 17,A -2.9012,B 0,C 0,E1 0.1598,E2 90.071} C_DIS
LIN {X -7.33,Y 1.8172,Z 17,A -2.961,B 0,C 0,E1 0.1598,E2 90.071} C_DIS
LIN {X -7.4811,Y 1.0283,Z 17,A -3.0001,B 0,C 0,E1 0.1598,E2 90.0712} C_DIS
LIN {X -7.5496,Y 0.228,Z 17,A -3.0364,B 0,C 0,E1 0.1598,E2 90.0712} C_DIS
LIN {X -7.502,Y -0.9105,Z 17,A -3.0823,B 0,C 0,E1 0.1598,E2 90.0708} C_DIS
LIN {X -7.3399,Y -1.7807,Z 17,A -3.1133,B 0,C 0,E1 0.1598,E2 90.0711} C_DIS
LIN {X -7.0338,Y -2.7671,Z 17,A -3.1435,B 0,C 0,E1 0.1598,E2 90.0709} C_DIS
LIN {X -6.5466,Y -3.7662,Z 17,A -3.1677,B 0,C 0,E1 0.1598,E2 90.0709} C_DIS
LIN {X -6.1126,Y -4.4367,Z 17,A -3.1803,B 0,C 0,E1 0.1598,E2 90.0711} C_DIS
LIN {X -5.6102,Y -5.0576,Z 17,A -3.1882,B 0,C 0,E1 0.1598,E2 90.0711} C_DIS
LIN {X -5.0447,Y -5.6217,Z 17,A -3.1913,B 0,C 0,E1 0.1598,E2 90.0711} C_DIS
LIN {X -4.423,Y -6.1231,Z 17,A -3.1897,B 0,C 0,E1 0.1598,E2 90.0711} C_DIS
LIN {X -3.7516,Y -6.5558,Z 17,A -3.1834,B 0,C 0,E1 0.1598,E2 90.0712} C_DIS
LIN {X -2.856,Y -6.9969,Z 17,A -3.1692,B 0,C 0,E1 0.1598,E2 90.0712} C_DIS
LIN {X -1.7073,Y -7.358,Z 17,A -3.1424,B 0,C 0,E1 0.1598,E2 90.0713} C_DIS
LIN {X -0.964,Y -7.4959,Z 17,A -3.1211,B 0,C 0,E1 0.1598,E2 90.0713} C_DIS
LIN {X 0.0486,Y -7.5544,Z 17,A -3.0864,B 0,C 0,E1 0.1598,E2 90.0715} C_DIS
Enddeposition()
LIN {X 0.0486,Y -7.5544,Z 17,A -3.0864,B 0,C 0,E1 0.1598,E2 90.0715} C_DIS
Startdeposition()
$VEL.CP = VEL_PRINT
LIN {X -0.5319,Y -8.4709,Z 17,A -3.1462,B 0,C 0,E1 0.1598,E2 90.0708} C_DIS
LIN {X -1.327,Y -8.3819,Z 17,A -3.1721,B 0,C 0,E1 0.1598,E2 90.0713} C_DIS
LIN {X -2.1104,Y -8.219,Z 17,A -3.1939,B 0,C 0,E1 0.1598,E2 90.0713} C_DIS
LIN {X -2.875,Y -7.9834,Z 17,A -3.212,B 0,C 0,E1 0.1598,E2 90.0713} C_DIS
LIN {X -3.6142,Y -7.6773,Z 17,A -3.2261,B 0,C 0,E1 0.1598,E2 90.0713} C_DIS
LIN {X -4.3214,Y -7.3031,Z 17,A -3.2362,B 0,C 0,E1 0.1598,E2 90.0712} C_DIS
LIN {X -4.9905,Y -6.8643,Z 17,A -3.2421,B 0,C 0,E1 0.1598,E2 90.0712} C_DIS
LIN {X -5.6156,Y -6.3646,Z 17,A -3.2439,B 0,C 0,E1 0.1598,E2 90.0712} C_DIS
LIN {X -6.4305,Y -5.5434,Z 17,A -3.2389,B 0,C 0,E1 0.1598,E2 90.0709} C_DIS
LIN {X -7.048,Y -4.7289,Z 17,A -3.2272,B 0,C 0,E1 0.1598,E2 90.0709} C_DIS
LIN {X -7.471,Y -4.0292,Z 17,A -3.2133,B 0,C 0,E1 0.1598,E2 90.071} C_DIS
LIN {X -7.9046,Y -3.1037,Z 17,A -3.1899,B 0,C 0,E1 0.1598,E2 90.0708} C_DIS
LIN {X -8.2047,Y -2.1842,Z 17,A -3.1622,B 0,C 0,E1 0.1598,E2 90.0709} C_DIS
LIN {X -8.4121,Y -1.1639,Z 17,A -3.1267,B 0,C 0,E1 0.1598,E2 90.0709} C_DIS
LIN {X -8.4897,Y 0.1333,Z 17,A -3.0747,B 0,C 0,E1 0.1598,E2 90.0707} C_DIS
LIN {X -8.4067,Y 1.1608,Z 17,A -3.0286,B 0,C 0,E1 0.1598,E2 90.071} C_DIS
LIN {X -8.2542,Y 1.9713,Z 17,A -2.989,B 0,C 0,E1 0.1598,E2 90.0712} C_DIS
LIN {X -8.024,Y 2.7632,Z 17,A -2.9472,B 0,C 0,E1 0.1598,E2 90.0713} C_DIS
LIN {X -7.7181,Y 3.5291,Z 17,A -2.9037,B 0,C 0,E1 0.1598,E2 90.0714} C_DIS
LIN {X -7.3393,Y 4.2618,Z 17,A -2.859,B 0,C 0,E1 0.1598,E2 90.0714} C_DIS
LIN {X -6.8914,Y 4.9543,Z 17,A -2.8133,B 0,C 0,E1 0.1598,E2 90.0716} C_DIS
LIN {X -6.3785,Y 5.6003,Z 17,A -2.7672,B 0,C 0,E1 0.1598,E2 90.0716} C_DIS
LIN {X -5.5474,Y 6.4271,Z 17,A -2.7016,B 0,C 0,E1 0.1598,E2 90.0716} C_DIS
LIN {X -4.7277,Y 7.049,Z 17,A -2.6453,B 0,C 0,E1 0.1598,E2 90.0719} C_DIS
LIN {X -4.0229,Y 7.4739,Z 17,A -2.6015,B 0,C 0,E1 0.1598,E2 90.072} C_DIS
LIN {X -3.2802,Y 7.8285,Z 17,A -2.5591,B 0,C 0,E1 0.1598,E2 90.0721} C_DIS
LIN {X -2.5067,Y 8.1098,Z 17,A -2.5187,B 0,C 0,E1 0.1598,E2 90.0721} C_DIS
LIN {X -1.7094,Y 8.314,Z 17,A -2.4807,B 0,C 0,E1 0.1598,E2 90.0722} C_DIS
LIN {X -0.8962,Y 8.4414,Z 17,A -2.4453,B 0,C 0,E1 0.1598,E2 90.0723} C_DIS
LIN {X -0.0744,Y 8.4875,Z 17,A -2.413,B 0,C 0,E1 0.1598,E2 90.0723} C_DIS
LIN {X 0.7478,Y 8.4538,Z 17,A -2.3841,B 0,C 0,E1 0.1598,E2 90.0723} C_DIS
LIN {X 1.5631,Y 8.3411,Z 17,A -2.3587,B 0,C 0,E1 0.1598,E2 90.0724} C_DIS
LIN {X 2.3637,Y 8.1504,Z 17,A -2.3372,B 0,C 0,E1 0.1598,E2 90.0724} C_DIS
LIN {X 3.1423,Y 7.8836,Z 17,A -2.3197,B 0,C 0,E1 0.1598,E2 90.0724} C_DIS
LIN {X 3.8913,Y 7.5424,Z 17,A -2.3065,B 0,C 0,E1 0.1598,E2 90.0724} C_DIS
LIN {X 4.6039,Y 7.1302,Z 17,A -2.2976,B 0,C 0,E1 0.1598,E2 90.0724} C_DIS
LIN {X 5.2733,Y 6.6512,Z 17,A -2.2931,B 0,C 0,E1 0.1598,E2 90.0724} C_DIS
LIN {X 6.1386,Y 5.865,Z 17,A -2.2943,B 0,C 0,E1 0.1598,E2 90.0721} C_DIS
LIN {X 6.789,Y 5.093,Z 17,A -2.3031,B 0,C 0,E1 0.1598,E2 90.0721} C_DIS
LIN {X 7.2435,Y 4.4257,Z 17,A -2.3147,B 0,C 0,E1 0.1598,E2 90.0722} C_DIS
LIN {X 7.6318,Y 3.7176,Z 17,A -2.3305,B 0,C 0,E1 0.1598,E2 90.0722} C_DIS
LIN {X 7.9506,Y 2.9756,Z 17,A -2.3502,B 0,C 0,E1 0.1598,E2 90.0722} C_DIS
LIN {X 8.1956,Y 2.2062,Z 17,A -2.3738,B 0,C 0,E1 0.1598,E2 90.0721} C_DIS
LIN {X 8.3686,Y 1.4174,Z 17,A -2.401,B 0,C 0,E1 0.1598,E2 90.0721} C_DIS
LIN {X 8.4818,Y 0.4145,Z 17,A -2.4392,B 0,C 0,E1 0.1598,E2 90.0717} C_DIS
LIN {X 8.4492,Y -0.801,Z 17,A -2.4918,B 0,C 0,E1 0.1598,E2 90.0714} C_DIS
LIN {X 8.246,Y -2.0254,Z 17,A -2.5514,B 0,C 0,E1 0.1598,E2 90.0714} C_DIS
LIN {X 7.9238,Y -3.0427,Z 17,A -2.6068,B 0,C 0,E1 0.1598,E2 90.0716} C_DIS
LIN {X 7.578,Y -3.8232,Z 17,A -2.6529,B 0,C 0,E1 0.1598,E2 90.0717} C_DIS
LIN {X 7.1549,Y -4.5647,Z 17,A -2.7,B 0,C 0,E1 0.1598,E2 90.0717} C_DIS
LIN {X 6.6606,Y -5.2607,Z 17,A -2.7478,B 0,C 0,E1 0.1598,E2 90.0717} C_DIS
LIN {X 5.9507,Y -6.0573,Z 17,A -2.8076,B 0,C 0,E1 0.1598,E2 90.0715} C_DIS
LIN {X 5.0713,Y -6.8053,Z 17,A -2.8717,B 0,C 0,E1 0.1598,E2 90.0715} C_DIS
LIN {X 4.4133,Y -7.2513,Z 17,A -2.915,B 0,C 0,E1 0.1598,E2 90.0715} C_DIS
LIN {X 3.7159,Y -7.6331,Z 17,A -2.9568,B 0,C 0,E1 0.1598,E2 90.0715} C_DIS
LIN {X 2.9853,Y -7.9467,Z 17,A -2.997,B 0,C 0,E1 0.1598,E2 90.0715} C_DIS
LIN {X 2.2286,Y -8.1904,Z 17,A -3.0351,B 0,C 0,E1 0.1598,E2 90.0715} C_DIS
LIN {X 1.4525,Y -8.3623,Z 17,A -3.0708,B 0,C 0,E1 0.1598,E2 90.0715} C_DIS
LIN {X 0.6638,Y -8.4606,Z 17,A -3.1039,B 0,C 0,E1 0.1598,E2 90.0715} C_DIS
LIN {X 0.6638,Y -8.4606,Z 17,A -3.1039,B 0,C 0,E1 0.1598,E2 90.0715} C_DIS
Enddeposition()
LIN {X 0.0003,Y -4.7569,Z 18,A -2.956,B 0,C 0,E1 0.1598,E2 90.0603} C_DIS
Startdeposition()
$VEL.CP = VEL_PRINT
LIN {X 0.0003,Y -4.7569,Z 18,A -2.9617,B 0,C 0,E1 0.1598,E2 90.0661} C_DIS
LIN {X 0.9387,Y -4.6571,Z 18,A -2.9279,B 0,C 0,E1 0.1598,E2 90.071} C_DIS
LIN {X 1.664,Y -4.448,Z 18,A -2.893,B 0,C 0,E1 0.1598,E2 90.0717} C_DIS
LIN {X 2.3471,Y -4.1277,Z 18,A -2.8543,B 0,C 0,E1 0.1598,E2 90.0717} C_DIS
LIN {X 3.0091,Y -3.6752,Z 18,A -2.8108,B 0,C 0,E1 0.1598,E2 90.0717} C_DIS
LIN {X 3.5213,Y -3.187,Z 18,A -2.7712,B 0,C 0,E1 0.1598,E2 90.0717} C_DIS
LIN {X 3.9814,Y -2.5888,Z 18,A -2.7289,B 0,C 0,E1 0.1598,E2 90.0717} C_DIS
LIN {X 4.3793,Y -1.8391,Z 18,A -2.6823,B 0,C 0,E1 0.1598,E2 90.0717} C_DIS
LIN {X 4.5934,Y -1.214,Z 18,A -2.648,B 0,C 0,E1 0.1598,E2 90.0718} C_DIS
LIN {X 4.7285,Y -0.4712,Z 18,A -2.6114,B 0,C 0,E1 0.1598,E2 90.0718} C_DIS
LIN {X 4.7428,Y 0.2836,Z 18,A -2.5788,B 0,C 0,E1 0.1598,E2 90.0718} C_DIS
LIN {X 4.6368,Y 1.0312,Z 18,A -2.551,B 0,C 0,E1 0.1598,E2 90.0718} C_DIS
LIN {X 4.4156,Y 1.7529,Z 18,A -2.5285,B 0,C 0,E1 0.1598,E2 90.0719} C_DIS
LIN {X 4.081,Y 2.4295,Z 18,A -2.5122,B 0,C 0,E1 0.1598,E2 90.0719} C_DIS
LIN {X 3.6449,Y 3.0454,Z 18,A -2.5022,B 0,C 0,E1 0.1598,E2 90.072} C_DIS
LIN {X 3.1171,Y 3.5851,Z 18,A -2.4988,B 0,C 0,E1 0.1598,E2 90.072} C_DIS
LIN {X 2.509,Y 4.032,Z 18,A -2.5023,B 0,C 0,E1 0.1598,E2 90.0721} C_DIS
LIN {X 1.839,Y 4.3794,Z 18,A -2.5124,B 0,C 0,E1 0.1598,E2 90.0721} C_DIS
LIN {X 1.1222,Y 4.6155,Z 18,A -2.5288,B 0,C 0,E1 0.1598,E2 90.0721} C_DIS
LIN {X 0.377,Y 4.735,Z 18,A -2.5513,B 0,C 0,E1 0.1598,E2 90.0721} C_DIS
LIN {X -0.3776,Y 4.734,Z 18,A -2.5792,B 0,C 0,E1 0.1598,E2 90.0721} C_DIS
LIN {X -1.1228,Y 4.6145,Z 18,A -2.6117,B 0,C 0,E1 0.1598,E2 90.0721} C_DIS
LIN {X -1.8401,Y 4.3797,Z 18,A -2.648,B 0,C 0,E1 0.1598,E2 90.0721} C_DIS
LIN {X -2.5113,Y 4.034,Z 18,A -2.6873,B 0,C 0,E1 0.1598,E2 90.0719} C_DIS
LIN {X -3.1174,Y 3.5839,Z 18,A -2.7286,B 0,C 0,E1 0.1598,E2 90.0719} C_DIS
LIN {X -3.6455,Y 3.0445,Z 18,A -2.7708,B 0,C 0,E1 0.1598,E2 90.0717} C_DIS
LIN {X -4.0815,Y 2.4286,Z 18,A -2.8128,B 0,C 0,E1 0.1598,E2 90.0717} C_DIS
LIN {X -4.414,Y 1.7512,Z 18,A -2.8536,B 0,C 0,E1 0.1598,E2 90.0715} C_DIS
LIN {X -4.6367,Y 1.0302,Z 18,A -2.8922,B 0,C 0,E1 0.1598,E2 90.0715} C_DIS
LIN {X -4.741,Y 0.2827,Z 18,A -2.9276,B 0,C 0,E1 0.1598,E2 90.0714} C_DIS
LIN {X -4.7256,Y -0.4719,Z 18,A -2.9588,B 0,C 0,E1 0.1598,E2 90.0714} C_DIS
LIN {X -4.5914,Y -1.2145,Z 18,A -2.9853,B 0,C 0,E1 0.1598,E2 90.0714} C_DIS
LIN {X -4.3408,Y -1.9264,Z 18,A -3.0061,B 0,C 0,E1 0.1598,E2 90.0713} C_DIS
LIN {X -3.9809,Y -2.5897,Z 18,A -3.021,B 0,C 0,E1 0.1598,E2 90.0713} C_DIS
LIN {X -3.5208,Y -3.1879,Z 18,A -3.0294,B 0,C 0,E1 0.1598,E2 90.0713} C_DIS
LIN {X -2.972,Y -3.7062,Z 18,A -3.0312,B 0,C 0,E1 0.1598,E2 90.0713} C_DIS
LIN {X -2.3474,Y -4.1296,Z 18,A -3.0262,B 0,C 0,E1 0.1598,E2 90.0714} C_DIS
LIN {X -1.664,Y -4.4505,Z 18,A -3.0147,B 0,C 0,E1 0.1598,E2 90.0714} C_DIS
LIN {X -0.938,Y -4.6576,Z 18,A -2.9969,B 0,C 0,E1 0.1598,E2 90.0716} C_DIS
LIN {X 0.0003,Y -4.7569,Z 18,A -2.9667,B 0,C 0,E1 0.1598,E2 90.0716} C_DIS
Enddeposition()
LIN {X 0.0003,Y -4.7569,Z 18,A -2.9667,B 0,C 0,E1 0.1598,E2 90.0716} C_DIS
Startdeposition()
$VEL.CP = VEL_PRINT
LIN {X -0.5996,Y -5.6514,Z 18,A -3.0262,B 0,C 0,E1 0.1598,E2 90.071} C_DIS
LIN {X -1.3863,Y -5.5122,Z 18,A -3.0497,B 0,C 0,E1 0.1598,E2 90.0715} C_DIS
LIN {X -2.4821,Y -5.1193,Z 18,A -3.0732,B 0,C 0,E1 0.1598,E2 90.0714} C_DIS
LIN {X -3.0018,Y -4.828,Z 18,A -3.08,B 0,C 0,E1 0.1598,E2 90.0714} C_DIS
LIN {X -3.6454,Y -4.363,Z 18,A -3.0839,B 0,C 0,E1 0.1598,E2 90.0714} C_DIS
LIN {X -4.2167,Y -3.8118,Z 18,A -3.0815,B 0,C 0,E1 0.1598,E2 90.0713} C_DIS
LIN {X -4.7052,Y -3.1863,Z 18,A -3.073,B 0,C 0,E1 0.1598,E2 90.0713} C_DIS
LIN {X -5.1034,Y -2.5,Z 18,A -3.0586,B 0,C 0,E1 0.1598,E2 90.0713} C_DIS
LIN {X -5.4017,Y -1.7646,Z 18,A -3.0384,B 0,C 0,E1 0.1598,E2 90.0713} C_DIS
LIN {X -5.5953,Y -0.995,Z 18,A -3.013,B 0,C 0,E1 0.1598,E2 90.0713} C_DIS
LIN {X -5.6801,Y -0.206,Z 18,A -2.9828,B 0,C 0,E1 0.1598,E2 90.0713} C_DIS
LIN {X -5.6538,Y 0.5874,Z 18,A -2.9484,B 0,C 0,E1 0.1598,E2 90.0713} C_DIS
LIN {X -5.5178,Y 1.3694,Z 18,A -2.9104,B 0,C 0,E1 0.1598,E2 90.0713} C_DIS
LIN {X -5.2705,Y 2.1236,Z 18,A -2.8695,B 0,C 0,E1 0.1598,E2 90.0715} C_DIS
LIN {X -4.9259,Y 2.8385,Z 18,A -2.8267,B 0,C 0,E1 0.1598,E2 90.0715} C_DIS
LIN {X -4.4828,Y 3.4973,Z 18,A -2.7826,B 0,C 0,E1 0.1598,E2 90.0716} C_DIS
LIN {X -3.9521,Y 4.088,Z 18,A -2.7382,B 0,C 0,E1 0.1598,E2 90.0717} C_DIS
LIN {X -3.3429,Y 4.597,Z 18,A -2.6943,B 0,C 0,E1 0.1598,E2 90.0719} C_DIS
LIN {X -2.3891,Y 5.1645,Z 18,A -2.6351,B 0,C 0,E1 0.1598,E2 90.0719} C_DIS
LIN {X -1.5132,Y 5.4852,Z 18,A -2.5894,B 0,C 0,E1 0.1598,E2 90.0721} C_DIS
LIN {X -0.4982,Y 5.662,Z 18,A -2.5445,B 0,C 0,E1 0.1598,E2 90.0721} C_DIS
LIN {X 0.326,Y 5.6752,Z 18,A -2.5136,B 0,C 0,E1 0.1598,E2 90.0722} C_DIS
LIN {X 1.1431,Y 5.5669,Z 18,A -2.488,B 0,C 0,E1 0.1598,E2 90.0722} C_DIS
LIN {X 1.9358,Y 5.3421,Z 18,A -2.4682,B 0,C 0,E1 0.1598,E2 90.0722} C_DIS
LIN {X 2.6888,Y 5.007,Z 18,A -2.4546,B 0,C 0,E1 0.1598,E2 90.0722} C_DIS
LIN {X 3.3854,Y 4.5662,Z 18,A -2.4476,B 0,C 0,E1 0.1598,E2 90.0722} C_DIS
LIN {X 4.011,Y 4.0291,Z 18,A -2.4472,B 0,C 0,E1 0.1598,E2 90.0722} C_DIS
LIN {X 4.5515,Y 3.4066,Z 18,A -2.4536,B 0,C 0,E1 0.1598,E2 90.0721} C_DIS
LIN {X 4.9965,Y 2.7124,Z 18,A -2.4666,B 0,C 0,E1 0.1598,E2 90.0721} C_DIS
LIN {X 5.336,Y 1.9611,Z 18,A -2.4859,B 0,C 0,E1 0.1598,E2 90.0719} C_DIS
LIN {X 5.561,Y 1.1681,Z 18,A -2.5113,B 0,C 0,E1 0.1598,E2 90.0719} C_DIS
LIN {X 5.672,Y 0.3516,Z 18,A -2.5418,B 0,C 0,E1 0.1598,E2 90.0719} C_DIS
LIN {X 5.6625,Y -0.4723,Z 18,A -2.5772,B 0,C 0,E1 0.1598,E2 90.0718} C_DIS
LIN {X 5.535,Y -1.2865,Z 18,A -2.6164,B 0,C 0,E1 0.1598,E2 90.0718} C_DIS
LIN {X 5.2922,Y -2.0741,Z 18,A -2.6588,B 0,C 0,E1 0.1598,E2 90.0717} C_DIS
LIN {X 4.9372,Y -2.8181,Z 18,A -2.7035,B 0,C 0,E1 0.1598,E2 90.0717} C_DIS
LIN {X 4.477,Y -3.5021,Z 18,A -2.7495,B 0,C 0,E1 0.1598,E2 90.0717} C_DIS
LIN {X 3.9238,Y -4.1134,Z 18,A -2.7959,B 0,C 0,E1 0.1598,E2 90.0717} C_DIS
LIN {X 3.2873,Y -4.6374,Z 18,A -2.8415,B 0,C 0,E1 0.1598,E2 90.0717} C_DIS
LIN {X 2.582,Y -5.0642,Z 18,A -2.8856,B 0,C 0,E1 0.1598,E2 90.0717} C_DIS
LIN {X 1.8223,Y -5.3843,Z 18,A -2.9271,B 0,C 0,E1 0.1598,E2 90.0717} C_DIS
LIN {X 1.0241,Y -5.5892,Z 18,A -2.9651,B 0,C 0,E1 0.1598,E2 90.0717} C_DIS
LIN {X 0.2049,Y -5.6785,Z 18,A -2.999,B 0,C 0,E1 0.1598,E2 90.0716} C_DIS
LIN {X 0.2049,Y -5.6785,Z 18,A -2.999,B 0,C 0,E1 0.1598,E2 90.0716} C_DIS
Enddeposition()
LIN {X 0.0244,Y -6.6219,Z 18,A -3.0446,B 0,C 0,E1 0.1598,E2 90.0703} C_DIS
Startdeposition()
$VEL.CP = VEL_PRINT
LIN {X 0.8954,Y -6.5591,Z 18,A -3.0111,B 0,C 0,E1 0.1598,E2 90.0715} C_DIS
LIN {X 1.9106,Y -6.3418,Z 18,A -2.9646,B 0,C 0,E1 0.1598,E2 90.0715} C_DIS
LIN {X 2.7991,Y -5.9988,Z 18,A -2.9175,B 0,C 0,E1 0.1598,E2 90.0716} C_DIS
LIN {X 3.469,Y -5.6359,Z 18,A -2.8774,B 0,C 0,E1 0.1598,E2 90.0716} C_DIS
LIN {X 4.0937,Y -5.2,Z 18,A -2.836,B 0,C 0,E1 0.1598,E2 90.0717} C_DIS
LIN {X 4.6641,Y -4.695,Z 18,A -2.7935,B 0,C 0,E1 0.1598,E2 90.0717} C_DIS
LIN {X 5.1727,Y -4.128,Z 18,A -2.7507,B 0,C 0,E1 0.1598,E2 90.0717} C_DIS
LIN {X 5.6158,Y -3.5082,Z 18,A -2.7081,B 0,C 0,E1 0.1598,E2 90.0717} C_DIS
LIN {X 5.9812,Y -2.8397,Z 18,A -2.6662,B 0,C 0,E1 0.1598,E2 90.0717} C_DIS
LIN {X 6.2658,Y -2.133,Z 18,A -2.6257,B 0,C 0,E1 0.1598,E2 90.0718} C_DIS
LIN {X 6.4693,Y -1.3988,Z 18,A -2.587,B 0,C 0,E1 0.1598,E2 90.0718} C_DIS
LIN {X 6.5867,Y -0.6461,Z 18,A -2.5507,B 0,C 0,E1 0.1598,E2 90.0718} C_DIS
LIN {X 6.6167,Y 0.115,Z 18,A -2.5172,B 0,C 0,E1 0.1598,E2 90.0718} C_DIS
LIN {X 6.5615,Y 0.8748,Z 18,A -2.4869,B 0,C 0,E1 0.1598,E2 90.0719} C_DIS
LIN {X 6.3374,Y 1.9247,Z 18,A -2.4503,B 0,C 0,E1 0.1598,E2 90.0717} C_DIS
LIN {X 6.0225,Y 2.7473,Z 18,A -2.4272,B 0,C 0,E1 0.1598,E2 90.072} C_DIS
LIN {X 5.6958,Y 3.3717,Z 18,A -2.4129,B 0,C 0,E1 0.1598,E2 90.0721} C_DIS
LIN {X 5.3066,Y 3.9592,Z 18,A -2.4023,B 0,C 0,E1 0.1598,E2 90.0721} C_DIS
LIN {X 4.8547,Y 4.4997,Z 18,A -2.3961,B 0,C 0,E1 0.1598,E2 90.0722} C_DIS
LIN {X 4.3481,Y 4.9894,Z 18,A -2.3941,B 0,C 0,E1 0.1598,E2 90.0722} C_DIS
LIN {X 3.7929,Y 5.4233,Z 18,A -2.3962,B 0,C 0,E1 0.1598,E2 90.0722} C_DIS
LIN {X 3.1956,Y 5.7971,Z 18,A -2.4024,B 0,C 0,E1 0.1598,E2 90.0722} C_DIS
LIN {X 2.5614,Y 6.1046,Z 18,A -2.4128,B 0,C 0,E1 0.1598,E2 90.0722} C_DIS
LIN {X 1.8981,Y 6.3424,Z 18,A -2.4272,B 0,C 0,E1 0.1598,E2 90.0722} C_DIS
LIN {X 1.213,Y 6.5074,Z 18,A -2.4456,B 0,C 0,E1 0.1598,E2 90.0722} C_DIS
LIN {X 0.5144,Y 6.5996,Z 18,A -2.4675,B 0,C 0,E1 0.1598,E2 90.0722} C_DIS
LIN {X -0.1901,Y 6.6162,Z 18,A -2.4928,B 0,C 0,E1 0.1598,E2 90.0722} C_DIS
LIN {X -0.8925,Y 6.5594,Z 18,A -2.5211,B 0,C 0,E1 0.1598,E2 90.0722} C_DIS
LIN {X -1.5848,Y 6.4287,Z 18,A -2.5521,B 0,C 0,E1 0.1598,E2 90.0722} C_DIS
LIN {X -2.2594,Y 6.2247,Z 18,A -2.5856,B 0,C 0,E1 0.1598,E2 90.0722} C_DIS
LIN {X -2.907,Y 5.9468,Z 18,A -2.6212,B 0,C 0,E1 0.1598,E2 90.072} C_DIS
LIN {X -3.5227,Y 5.604,Z 18,A -2.6584,B 0,C 0,E1 0.1598,E2 90.072} C_DIS
LIN {X -4.0994,Y 5.1992,Z 18,A -2.6967,B 0,C 0,E1 0.1598,E2 90.0719} C_DIS
LIN {X -4.6282,Y 4.7335,Z 18,A -2.7358,B 0,C 0,E1 0.1598,E2 90.0719} C_DIS
LIN {X -5.1052,Y 4.2147,Z 18,A -2.7752,B 0,C 0,E1 0.1598,E2 90.0717} C_DIS
LIN {X -5.5234,Y 3.6474,Z 18,A -2.8145,B 0,C 0,E1 0.1598,E2 90.0717} C_DIS
LIN {X -5.8802,Y 3.0397,Z 18,A -2.8533,B 0,C 0,E1 0.1598,E2 90.0716} C_DIS
LIN {X -6.17,Y 2.3976,Z 18,A -2.891,B 0,C 0,E1 0.1598,E2 90.0716} C_DIS
LIN {X -6.3895,Y 1.728,Z 18,A -2.9273,B 0,C 0,E1 0.1598,E2 90.0714} C_DIS
LIN {X -6.5375,Y 1.0391,Z 18,A -2.9618,B 0,C 0,E1 0.1598,E2 90.0714} C_DIS
LIN {X -6.6118,Y 0.3385,Z 18,A -2.994,B 0,C 0,E1 0.1598,E2 90.0714} C_DIS
LIN {X -6.6089,Y -0.3662,Z 18,A -3.0236,B 0,C 0,E1 0.1598,E2 90.0713} C_DIS
LIN {X -6.5344,Y -1.0669,Z 18,A -3.0504,B 0,C 0,E1 0.1598,E2 90.0713} C_DIS
LIN {X -6.3836,Y -1.7555,Z 18,A -3.0739,B 0,C 0,E1 0.1598,E2 90.0713} C_DIS
LIN {X -6.1603,Y -2.4239,Z 18,A -3.094,B 0,C 0,E1 0.1598,E2 90.0713} C_DIS
LIN {X -5.867,Y -3.0647,Z 18,A -3.1103,B 0,C 0,E1 0.1598,E2 90.0713} C_DIS
LIN {X -5.5081,Y -3.6712,Z 18,A -3.1227,B 0,C 0,E1 0.1598,E2 90.0713} C_DIS
LIN {X -4.8752,Y -4.4838,Z 18,A -3.1336,B 0,C 0,E1 0.1598,E2 90.0711} C_DIS
LIN {X -4.1702,Y -5.1409,Z 18,A -3.1357,B 0,C 0,E1 0.1598,E2 90.0711} C_DIS
LIN {X -3.2818,Y -5.7535,Z 18,A -3.129,B 0,C 0,E1 0.1598,E2 90.0712} C_DIS
LIN {X -2.5037,Y -6.1284,Z 18,A -3.1164,B 0,C 0,E1 0.1598,E2 90.0713} C_DIS
LIN {X -1.8516,Y -6.3565,Z 18,A -3.1022,B 0,C 0,E1 0.1598,E2 90.0714} C_DIS
LIN {X -1.1787,Y -6.5136,Z 18,A -3.0842,B 0,C 0,E1 0.1598,E2 90.0714} C_DIS
LIN {X -0.4934,Y -6.6,Z 18,A -3.0627,B 0,C 0,E1 0.1598,E2 90.0714} C_DIS
LIN {X -0.4934,Y -6.6,Z 18,A -3.0627,B 0,C 0,E1 0.1598,E2 90.0714} C_DIS
Enddeposition()
LIN {X 0.0091,Y -7.5541,Z 18,A -3.0838,B 0,C 0,E1 0.1598,E2 90.0703} C_DIS
Startdeposition()
$VEL.CP = VEL_PRINT
LIN {X -1.3127,Y -7.4428,Z 18,A -3.1286,B 0,C 0,E1 0.1598,E2 90.0713} C_DIS
LIN {X -2.4745,Y -7.1364,Z 18,A -3.1582,B 0,C 0,E1 0.1598,E2 90.0713} C_DIS
LIN {X -3.582,Y -6.6539,Z 18,A -3.1784,B 0,C 0,E1 0.1598,E2 90.0713} C_DIS
LIN {X -4.425,Y -6.122,Z 18,A -3.1868,B 0,C 0,E1 0.1598,E2 90.0712} C_DIS
LIN {X -5.0453,Y -5.621,Z 18,A -3.1883,B 0,C 0,E1 0.1598,E2 90.0712} C_DIS
LIN {X -5.6097,Y -5.0577,Z 18,A -3.1852,B 0,C 0,E1 0.1598,E2 90.0712} C_DIS
LIN {X -6.1116,Y -4.4381,Z 18,A -3.1774,B 0,C 0,E1 0.1598,E2 90.0712} C_DIS
LIN {X -6.5452,Y -3.7689,Z 18,A -3.1651,B 0,C 0,E1 0.1598,E2 90.0712} C_DIS
LIN {X -7.0354,Y -2.7626,Z 18,A -3.1403,B 0,C 0,E1 0.1598,E2 90.0709} C_DIS
LIN {X -7.3501,Y -1.7609,Z 18,A -3.1096,B 0,C 0,E1 0.1598,E2 90.0709} C_DIS
LIN {X -7.5402,Y -0.5022,Z 18,A -3.0632,B 0,C 0,E1 0.1598,E2 90.0706} C_DIS
LIN {X -7.5156,Y 0.7564,Z 18,A -3.0092,B 0,C 0,E1 0.1598,E2 90.0706} C_DIS
LIN {X -7.407,Y 1.4978,Z 18,A -2.9744,B 0,C 0,E1 0.1598,E2 90.0712} C_DIS
LIN {X -7.0341,Y 2.7646,Z 18,A -2.9069,B 0,C 0,E1 0.1598,E2 90.0708} C_DIS
LIN {X -6.6264,Y 3.6319,Z 18,A -2.8558,B 0,C 0,E1 0.1598,E2 90.0714} C_DIS
LIN {X -6.0559,Y 4.5209,Z 18,A -2.7973,B 0,C 0,E1 0.1598,E2 90.0714} C_DIS
LIN {X -5.3845,Y 5.2971,Z 18,A -2.7399,B 0,C 0,E1 0.1598,E2 90.0716} C_DIS
LIN {X -4.5196,Y 6.0569,Z 18,A -2.676,B 0,C 0,E1 0.1598,E2 90.0717} C_DIS
LIN {X -3.5803,Y 6.6505,Z 18,A -2.6164,B 0,C 0,E1 0.1598,E2 90.0719} C_DIS
LIN {X -2.5671,Y 7.1073,Z 18,A -2.5598,B 0,C 0,E1 0.1598,E2 90.072} C_DIS
LIN {X -1.447,Y 7.4177,Z 18,A -2.5054,B 0,C 0,E1 0.1598,E2 90.0722} C_DIS
LIN {X -0.3542,Y 7.5451,Z 18,A -2.4597,B 0,C 0,E1 0.1598,E2 90.0722} C_DIS
LIN {X 0.8213,Y 7.5121,Z 18,A -2.4177,B 0,C 0,E1 0.1598,E2 90.0723} C_DIS
LIN {X 1.8118,Y 7.3369,Z 18,A -2.3886,B 0,C 0,E1 0.1598,E2 90.0723} C_DIS
LIN {X 2.9085,Y 6.9745,Z 18,A -2.3634,B 0,C 0,E1 0.1598,E2 90.0723} C_DIS
LIN {X 4.1539,Y 6.3146,Z 18,A -2.3451,B 0,C 0,E1 0.1598,E2 90.0722} C_DIS
LIN {X 4.9972,Y 5.6651,Z 18,A -2.3416,B 0,C 0,E1 0.1598,E2 90.0722} C_DIS
LIN {X 5.8,Y 4.8443,Z 18,A -2.3466,B 0,C 0,E1 0.1598,E2 90.072} C_DIS
LIN {X 6.4946,Y 3.8575,Z 18,A -2.3627,B 0,C 0,E1 0.1598,E2 90.0718} C_DIS
LIN {X 6.8454,Y 3.202,Z 18,A -2.3778,B 0,C 0,E1 0.1598,E2 90.072} C_DIS
LIN {X 7.3042,Y 1.9372,Z 18,A -2.4142,B 0,C 0,E1 0.1598,E2 90.0715} C_DIS
LIN {X 7.492,Y 0.9991,Z 18,A -2.4474,B 0,C 0,E1 0.1598,E2 90.0718} C_DIS
LIN {X 7.5582,Y -0.0272,Z 18,A -2.4885,B 0,C 0,E1 0.1598,E2 90.0717} C_DIS
LIN {X 7.4845,Y -1.0125,Z 18,A -2.5332,B 0,C 0,E1 0.1598,E2 90.0717} C_DIS
LIN {X 7.339,Y -1.7893,Z 18,A -2.5717,B 0,C 0,E1 0.1598,E2 90.0718} C_DIS
LIN {X 7.0463,Y -2.733,Z 18,A -2.6224,B 0,C 0,E1 0.1598,E2 90.0715} C_DIS
LIN {X 6.3182,Y -4.1487,Z 18,A -2.7087,B 0,C 0,E1 0.1598,E2 90.0708} C_DIS
LIN {X 5.6867,Y -4.9686,Z 18,A -2.7676,B 0,C 0,E1 0.1598,E2 90.0715} C_DIS
LIN {X 5.1096,Y -5.5622,Z 18,A -2.8142,B 0,C 0,E1 0.1598,E2 90.0716} C_DIS
LIN {X 4.4699,Y -6.088,Z 18,A -2.86,B 0,C 0,E1 0.1598,E2 90.0716} C_DIS
LIN {X 3.7768,Y -6.5408,Z 18,A -2.9047,B 0,C 0,E1 0.1598,E2 90.0716} C_DIS
LIN {X 2.7459,Y -7.0416,Z 18,A -2.9638,B 0,C 0,E1 0.1598,E2 90.0716} C_DIS
LIN {X 1.5393,Y -7.3983,Z 18,A -3.0232,B 0,C 0,E1 0.1598,E2 90.0715} C_DIS
LIN {X 0.5277,Y -7.5336,Z 18,A -3.0661,B 0,C 0,E1 0.1598,E2 90.0715} C_DIS
LIN {X 0.5277,Y -7.5336,Z 18,A -3.0661,B 0,C 0,E1 0.1598,E2 90.0715} C_DIS
Enddeposition()
LIN {X 0.0339,Y -8.4915,Z 18,A -3.1239,B 0,C 0,E1 0.1598,E2 90.0702} C_DIS
Startdeposition()
$VEL.CP = VEL_PRINT
LIN {X 1.0792,Y -8.419,Z 18,A -3.0836,B 0,C 0,E1 0.1598,E2 90.0714} C_DIS
LIN {X 1.9043,Y -8.2711,Z 18,A -3.0471,B 0,C 0,E1 0.1598,E2 90.0715} C_DIS
LIN {X 2.7109,Y -8.0428,Z 18,A -3.0079,B 0,C 0,E1 0.1598,E2 90.0715} C_DIS
LIN {X 3.491,Y -7.7361,Z 18,A -2.9662,B 0,C 0,E1 0.1598,E2 90.0715} C_DIS
LIN {X 4.2372,Y -7.3541,Z 18,A -2.9226,B 0,C 0,E1 0.1598,E2 90.0716} C_DIS
LIN {X 4.9421,Y -6.9004,Z 18,A -2.8774,B 0,C 0,E1 0.1598,E2 90.0716} C_DIS
LIN {X 5.599,Y -6.3796,Z 18,A -2.8311,B 0,C 0,E1 0.1598,E2 90.0716} C_DIS
LIN {X 6.4319,Y -5.5419,Z 18,A -2.7647,B 0,C 0,E1 0.1598,E2 90.0716} C_DIS
LIN {X 7.0727,Y -4.6914,Z 18,A -2.705,B 0,C 0,E1 0.1598,E2 90.0716} C_DIS
LIN {X 7.5074,Y -3.9588,Z 18,A -2.658,B 0,C 0,E1 0.1598,E2 90.0717} C_DIS
LIN {X 7.8664,Y -3.1864,Z 18,A -2.6119,B 0,C 0,E1 0.1598,E2 90.0717} C_DIS
LIN {X 8.1459,Y -2.3818,Z 18,A -2.5673,B 0,C 0,E1 0.1598,E2 90.0717} C_DIS
LIN {X 8.3428,Y -1.5532,Z 18,A -2.5248,B 0,C 0,E1 0.1598,E2 90.0718} C_DIS
LIN {X 8.4576,Y -0.709,Z 18,A -2.4847,B 0,C 0,E1 0.1598,E2 90.0718} C_DIS
LIN {X 8.4866,Y 0.1424,Z 18,A -2.4474,B 0,C 0,E1 0.1598,E2 90.0719} C_DIS
LIN {X 8.4291,Y 0.9923,Z 18,A -2.4133,B 0,C 0,E1 0.1598,E2 90.0719} C_DIS
LIN {X 8.2867,Y 1.8322,Z 18,A -2.3829,B 0,C 0,E1 0.1598,E2 90.0719} C_DIS
LIN {X 8.0607,Y 2.6535,Z 18,A -2.3563,B 0,C 0,E1 0.1598,E2 90.072} C_DIS
LIN {X 7.7542,Y 3.4483,Z 18,A -2.3338,B 0,C 0,E1 0.1598,E2 90.072} C_DIS
LIN {X 7.3695,Y 4.2084,Z 18,A -2.3157,B 0,C 0,E1 0.1598,E2 90.0721} C_DIS
LIN {X 6.9107,Y 4.9262,Z 18,A -2.3022,B 0,C 0,E1 0.1598,E2 90.0721} C_DIS
LIN {X 6.3825,Y 5.5946,Z 18,A -2.2934,B 0,C 0,E1 0.1598,E2 90.0722} C_DIS
LIN {X 5.6345,Y 6.3526,Z 18,A -2.2887,B 0,C 0,E1 0.1598,E2 90.0722} C_DIS
LIN {X 4.707,Y 7.063,Z 18,A -2.2929,B 0,C 0,E1 0.1598,E2 90.0722} C_DIS
LIN {X 4.0005,Y 7.4857,Z 18,A -2.3013,B 0,C 0,E1 0.1598,E2 90.0724} C_DIS
LIN {X 3.2565,Y 7.8381,Z 18,A -2.3138,B 0,C 0,E1 0.1598,E2 90.0724} C_DIS
LIN {X 2.482,Y 8.1174,Z 18,A -2.3307,B 0,C 0,E1 0.1598,E2 90.0724} C_DIS
LIN {X 1.6839,Y 8.32,Z 18,A -2.3516,B 0,C 0,E1 0.1598,E2 90.0724} C_DIS
LIN {X 0.8698,Y 8.4437,Z 18,A -2.3764,B 0,C 0,E1 0.1598,E2 90.0724} C_DIS
LIN {X 0.0476,Y 8.4878,Z 18,A -2.4049,B 0,C 0,E1 0.1598,E2 90.0724} C_DIS
LIN {X -0.7749,Y 8.451,Z 18,A -2.4369,B 0,C 0,E1 0.1598,E2 90.0724} C_DIS
LIN {X -1.5901,Y 8.3358,Z 18,A -2.4718,B 0,C 0,E1 0.1598,E2 90.0723} C_DIS
LIN {X -2.3904,Y 8.1425,Z 18,A -2.5095,B 0,C 0,E1 0.1598,E2 90.0723} C_DIS
LIN {X -3.1682,Y 7.8727,Z 18,A -2.5496,B 0,C 0,E1 0.1598,E2 90.0721} C_DIS
LIN {X -3.9164,Y 7.5288,Z 18,A -2.5917,B 0,C 0,E1 0.1598,E2 90.0721} C_DIS
LIN {X -4.6278,Y 7.1142,Z 18,A -2.6354,B 0,C 0,E1 0.1598,E2 90.072} C_DIS
LIN {X -5.2958,Y 6.6328,Z 18,A -2.6803,B 0,C 0,E1 0.1598,E2 90.0719} C_DIS
LIN {X -6.0621,Y 5.9456,Z 18,A -2.7374,B 0,C 0,E1 0.1598,E2 90.0717} C_DIS
LIN {X -6.8085,Y 5.0674,Z 18,A -2.8018,B 0,C 0,E1 0.1598,E2 90.0714} C_DIS
LIN {X -7.2571,Y 4.403,Z 18,A -2.8465,B 0,C 0,E1 0.1598,E2 90.0715} C_DIS
LIN {X -7.6407,Y 3.6991,Z 18,A -2.8902,B 0,C 0,E1 0.1598,E2 90.0715} C_DIS
LIN {X -7.956,Y 2.9619,Z 18,A -2.9328,B 0,C 0,E1 0.1598,E2 90.0714} C_DIS
LIN {X -8.1982,Y 2.1976,Z 18,A -2.9739,B 0,C 0,E1 0.1598,E2 90.0714} C_DIS
LIN {X -8.369,Y 1.4144,Z 18,A -3.0132,B 0,C 0,E1 0.1598,E2 90.0712} C_DIS
LIN {X -8.4815,Y 0.4187,Z 18,A -3.059,B 0,C 0,E1 0.1598,E2 90.0709} C_DIS
LIN {X -8.4814,Y -0.4215,Z 18,A -3.0946,B 0,C 0,E1 0.1598,E2 90.0711} C_DIS
LIN {X -8.3319,Y -1.6176,Z 18,A -3.139,B 0,C 0,E1 0.1598,E2 90.0706} C_DIS
LIN {X -8.1482,Y -2.3903,Z 18,A -3.1652,B 0,C 0,E1 0.1598,E2 90.0709} C_DIS
LIN {X -7.7463,Y -3.4691,Z 18,A -3.1957,B 0,C 0,E1 0.1598,E2 90.0707} C_DIS
LIN {X -7.3625,Y -4.2229,Z 18,A -3.2138,B 0,C 0,E1 0.1598,E2 90.071} C_DIS
LIN {X -6.9057,Y -4.9348,Z 18,A -3.2271,B 0,C 0,E1 0.1598,E2 90.071} C_DIS
LIN {X -6.3805,Y -5.5978,Z 18,A -3.2359,B 0,C 0,E1 0.1598,E2 90.071} C_DIS
LIN {X -5.5374,Y -6.4356,Z 18,A -3.2402,B 0,C 0,E1 0.1598,E2 90.071} C_DIS
LIN {X -4.7847,Y -7.0111,Z 18,A -3.2371,B 0,C 0,E1 0.1598,E2 90.071} C_DIS
Enddeposition()
END
